(* IEC 61131-3 sources: TA/Tests/RetainTest/Man (part 20) *)

    RETAINTEST_NONRETAIN_STRUCTUREARRAYARRAY.ARRAYARRAY_USINT[2][0] := RETAINTEST_NONRETAIN_STRUCTUREARRAYARRAY.ARRAYARRAY_USINT[2][0] + 1;
    RETAINTEST_NONRETAIN_STRUCTUREARRAYARRAY.ARRAYARRAY_USINT[2][1] := RETAINTEST_NONRETAIN_STRUCTUREARRAYARRAY.ARRAYARRAY_USINT[2][1] + 1;
    RETAINTEST_NONRETAIN_STRUCTUREARRAYARRAY.ARRAYARRAY_USINT[2][2] := RETAINTEST_NONRETAIN_STRUCTUREARRAYARRAY.ARRAYARRAY_USINT[2][2] + 1;
    RETAINTEST_NONRETAIN_STRUCTUREARRAYARRAY.ARRAYARRAY_USINT[2][3] := RETAINTEST_NONRETAIN_STRUCTUREARRAYARRAY.ARRAYARRAY_USINT[2][3] + 1;
    RETAINTEST_NONRETAIN_STRUCTUREARRAYARRAY.ARRAYARRAY_USINT[2][4] := RETAINTEST_NONRETAIN_STRUCTUREARRAYARRAY.ARRAYARRAY_USINT[2][4] + 1;
    RETAINTEST_NONRETAIN_STRUCTUREARRAYARRAY.ARRAYARRAY_USINT[2][5] := RETAINTEST_NONRETAIN_STRUCTUREARRAYARRAY.ARRAYARRAY_USINT[2][5] + 1;
    RETAINTEST_NONRETAIN_STRUCTUREARRAYARRAY.ARRAYARRAY_USINT[2][6] := RETAINTEST_NONRETAIN_STRUCTUREARRAYARRAY.ARRAYARRAY_USINT[2][6] + 1;
    RETAINTEST_NONRETAIN_STRUCTUREARRAYARRAY.ARRAYARRAY_USINT[2][7] := RETAINTEST_NONRETAIN_STRUCTUREARRAYARRAY.ARRAYARRAY_USINT[2][7] + 1;
    RETAINTEST_NONRETAIN_STRUCTUREARRAYARRAY.ARRAYARRAY_USINT[2][8] := RETAINTEST_NONRETAIN_STRUCTUREARRAYARRAY.ARRAYARRAY_USINT[2][8] + 1;
    RETAINTEST_NONRETAIN_STRUCTUREARRAYARRAY.ARRAYARRAY_USINT[2][9] := RETAINTEST_NONRETAIN_STRUCTUREARRAYARRAY.ARRAYARRAY_USINT[2][9] + 1;

    RETAINTEST_NONRETAIN_STRUCTUREARRAYARRAY.ARRAYARRAY_USINT[3][0] := RETAINTEST_NONRETAIN_STRUCTUREARRAYARRAY.ARRAYARRAY_USINT[3][0] + 1;
    RETAINTEST_NONRETAIN_STRUCTUREARRAYARRAY.ARRAYARRAY_USINT[3][1] := RETAINTEST_NONRETAIN_STRUCTUREARRAYARRAY.ARRAYARRAY_USINT[3][1] + 1;
    RETAINTEST_NONRETAIN_STRUCTUREARRAYARRAY.ARRAYARRAY_USINT[3][2] := RETAINTEST_NONRETAIN_STRUCTUREARRAYARRAY.ARRAYARRAY_USINT[3][2] + 1;
    RETAINTEST_NONRETAIN_STRUCTUREARRAYARRAY.ARRAYARRAY_USINT[3][3] := RETAINTEST_NONRETAIN_STRUCTUREARRAYARRAY.ARRAYARRAY_USINT[3][3] + 1;
    RETAINTEST_NONRETAIN_STRUCTUREARRAYARRAY.ARRAYARRAY_USINT[3][4] := RETAINTEST_NONRETAIN_STRUCTUREARRAYARRAY.ARRAYARRAY_USINT[3][4] + 1;
    RETAINTEST_NONRETAIN_STRUCTUREARRAYARRAY.ARRAYARRAY_USINT[3][5] := RETAINTEST_NONRETAIN_STRUCTUREARRAYARRAY.ARRAYARRAY_USINT[3][5] + 1;
    RETAINTEST_NONRETAIN_STRUCTUREARRAYARRAY.ARRAYARRAY_USINT[3][6] := RETAINTEST_NONRETAIN_STRUCTUREARRAYARRAY.ARRAYARRAY_USINT[3][6] + 1;
    RETAINTEST_NONRETAIN_STRUCTUREARRAYARRAY.ARRAYARRAY_USINT[3][7] := RETAINTEST_NONRETAIN_STRUCTUREARRAYARRAY.ARRAYARRAY_USINT[3][7] + 1;
    RETAINTEST_NONRETAIN_STRUCTUREARRAYARRAY.ARRAYARRAY_USINT[3][8] := RETAINTEST_NONRETAIN_STRUCTUREARRAYARRAY.ARRAYARRAY_USINT[3][8] + 1;
    RETAINTEST_NONRETAIN_STRUCTUREARRAYARRAY.ARRAYARRAY_USINT[3][9] := RETAINTEST_NONRETAIN_STRUCTUREARRAYARRAY.ARRAYARRAY_USINT[3][9] + 1;

    RETAINTEST_NONRETAIN_STRUCTUREARRAYARRAY.ARRAYARRAY_USINT[4][0] := RETAINTEST_NONRETAIN_STRUCTUREARRAYARRAY.ARRAYARRAY_USINT[4][0] + 1;
    RETAINTEST_NONRETAIN_STRUCTUREARRAYARRAY.ARRAYARRAY_USINT[4][1] := RETAINTEST_NONRETAIN_STRUCTUREARRAYARRAY.ARRAYARRAY_USINT[4][1] + 1;
    RETAINTEST_NONRETAIN_STRUCTUREARRAYARRAY.ARRAYARRAY_USINT[4][2] := RETAINTEST_NONRETAIN_STRUCTUREARRAYARRAY.ARRAYARRAY_USINT[4][2] + 1;
    RETAINTEST_NONRETAIN_STRUCTUREARRAYARRAY.ARRAYARRAY_USINT[4][3] := RETAINTEST_NONRETAIN_STRUCTUREARRAYARRAY.ARRAYARRAY_USINT[4][3] + 1;
    RETAINTEST_NONRETAIN_STRUCTUREARRAYARRAY.ARRAYARRAY_USINT[4][4] := RETAINTEST_NONRETAIN_STRUCTUREARRAYARRAY.ARRAYARRAY_USINT[4][4] + 1;
    RETAINTEST_NONRETAIN_STRUCTUREARRAYARRAY.ARRAYARRAY_USINT[4][5] := RETAINTEST_NONRETAIN_STRUCTUREARRAYARRAY.ARRAYARRAY_USINT[4][5] + 1;
    RETAINTEST_NONRETAIN_STRUCTUREARRAYARRAY.ARRAYARRAY_USINT[4][6] := RETAINTEST_NONRETAIN_STRUCTUREARRAYARRAY.ARRAYARRAY_USINT[4][6] + 1;
    RETAINTEST_NONRETAIN_STRUCTUREARRAYARRAY.ARRAYARRAY_USINT[4][7] := RETAINTEST_NONRETAIN_STRUCTUREARRAYARRAY.ARRAYARRAY_USINT[4][7] + 1;
    RETAINTEST_NONRETAIN_STRUCTUREARRAYARRAY.ARRAYARRAY_USINT[4][8] := RETAINTEST_NONRETAIN_STRUCTUREARRAYARRAY.ARRAYARRAY_USINT[4][8] + 1;
    RETAINTEST_NONRETAIN_STRUCTUREARRAYARRAY.ARRAYARRAY_USINT[4][9] := RETAINTEST_NONRETAIN_STRUCTUREARRAYARRAY.ARRAYARRAY_USINT[4][9] + 1;

    RETAINTEST_NONRETAIN_STRUCTUREARRAYARRAY.ARRAYARRAY_USINT[5][0] := RETAINTEST_NONRETAIN_STRUCTUREARRAYARRAY.ARRAYARRAY_USINT[5][0] + 1;
    RETAINTEST_NONRETAIN_STRUCTUREARRAYARRAY.ARRAYARRAY_USINT[5][1] := RETAINTEST_NONRETAIN_STRUCTUREARRAYARRAY.ARRAYARRAY_USINT[5][1] + 1;
    RETAINTEST_NONRETAIN_STRUCTUREARRAYARRAY.ARRAYARRAY_USINT[5][2] := RETAINTEST_NONRETAIN_STRUCTUREARRAYARRAY.ARRAYARRAY_USINT[5][2] + 1;
    RETAINTEST_NONRETAIN_STRUCTUREARRAYARRAY.ARRAYARRAY_USINT[5][3] := RETAINTEST_NONRETAIN_STRUCTUREARRAYARRAY.ARRAYARRAY_USINT[5][3] + 1;
    RETAINTEST_NONRETAIN_STRUCTUREARRAYARRAY.ARRAYARRAY_USINT[5][4] := RETAINTEST_NONRETAIN_STRUCTUREARRAYARRAY.ARRAYARRAY_USINT[5][4] + 1;
    RETAINTEST_NONRETAIN_STRUCTUREARRAYARRAY.ARRAYARRAY_USINT[5][5] := RETAINTEST_NONRETAIN_STRUCTUREARRAYARRAY.ARRAYARRAY_USINT[5][5] + 1;
    RETAINTEST_NONRETAIN_STRUCTUREARRAYARRAY.ARRAYARRAY_USINT[5][6] := RETAINTEST_NONRETAIN_STRUCTUREARRAYARRAY.ARRAYARRAY_USINT[5][6] + 1;
    RETAINTEST_NONRETAIN_STRUCTUREARRAYARRAY.ARRAYARRAY_USINT[5][7] := RETAINTEST_NONRETAIN_STRUCTUREARRAYARRAY.ARRAYARRAY_USINT[5][7] + 1;
    RETAINTEST_NONRETAIN_STRUCTUREARRAYARRAY.ARRAYARRAY_USINT[5][8] := RETAINTEST_NONRETAIN_STRUCTUREARRAYARRAY.ARRAYARRAY_USINT[5][8] + 1;
    RETAINTEST_NONRETAIN_STRUCTUREARRAYARRAY.ARRAYARRAY_USINT[5][9] := RETAINTEST_NONRETAIN_STRUCTUREARRAYARRAY.ARRAYARRAY_USINT[5][9] + 1;

    RETAINTEST_NONRETAIN_STRUCTUREARRAYARRAY.ARRAYARRAY_USINT[6][0] := RETAINTEST_NONRETAIN_STRUCTUREARRAYARRAY.ARRAYARRAY_USINT[6][0] + 1;
    RETAINTEST_NONRETAIN_STRUCTUREARRAYARRAY.ARRAYARRAY_USINT[6][1] := RETAINTEST_NONRETAIN_STRUCTUREARRAYARRAY.ARRAYARRAY_USINT[6][1] + 1;
    RETAINTEST_NONRETAIN_STRUCTUREARRAYARRAY.ARRAYARRAY_USINT[6][2] := RETAINTEST_NONRETAIN_STRUCTUREARRAYARRAY.ARRAYARRAY_USINT[6][2] + 1;
    RETAINTEST_NONRETAIN_STRUCTUREARRAYARRAY.ARRAYARRAY_USINT[6][3] := RETAINTEST_NONRETAIN_STRUCTUREARRAYARRAY.ARRAYARRAY_USINT[6][3] + 1;
    RETAINTEST_NONRETAIN_STRUCTUREARRAYARRAY.ARRAYARRAY_USINT[6][4] := RETAINTEST_NONRETAIN_STRUCTUREARRAYARRAY.ARRAYARRAY_USINT[6][4] + 1;
    RETAINTEST_NONRETAIN_STRUCTUREARRAYARRAY.ARRAYARRAY_USINT[6][5] := RETAINTEST_NONRETAIN_STRUCTUREARRAYARRAY.ARRAYARRAY_USINT[6][5] + 1;
    RETAINTEST_NONRETAIN_STRUCTUREARRAYARRAY.ARRAYARRAY_USINT[6][6] := RETAINTEST_NONRETAIN_STRUCTUREARRAYARRAY.ARRAYARRAY_USINT[6][6] + 1;
    RETAINTEST_NONRETAIN_STRUCTUREARRAYARRAY.ARRAYARRAY_USINT[6][7] := RETAINTEST_NONRETAIN_STRUCTUREARRAYARRAY.ARRAYARRAY_USINT[6][7] + 1;
    RETAINTEST_NONRETAIN_STRUCTUREARRAYARRAY.ARRAYARRAY_USINT[6][8] := RETAINTEST_NONRETAIN_STRUCTUREARRAYARRAY.ARRAYARRAY_USINT[6][8] + 1;
    RETAINTEST_NONRETAIN_STRUCTUREARRAYARRAY.ARRAYARRAY_USINT[6][9] := RETAINTEST_NONRETAIN_STRUCTUREARRAYARRAY.ARRAYARRAY_USINT[6][9] + 1;

    RETAINTEST_NONRETAIN_STRUCTUREARRAYARRAY.ARRAYARRAY_USINT[7][0] := RETAINTEST_NONRETAIN_STRUCTUREARRAYARRAY.ARRAYARRAY_USINT[6][0];
    RETAINTEST_NONRETAIN_STRUCTUREARRAYARRAY.ARRAYARRAY_USINT[7][1] := RETAINTEST_NONRETAIN_STRUCTUREARRAYARRAY.ARRAYARRAY_USINT[6][1];
    RETAINTEST_NONRETAIN_STRUCTUREARRAYARRAY.ARRAYARRAY_USINT[7][2] := RETAINTEST_NONRETAIN_STRUCTUREARRAYARRAY.ARRAYARRAY_USINT[6][2];
    RETAINTEST_NONRETAIN_STRUCTUREARRAYARRAY.ARRAYARRAY_USINT[7][3] := RETAINTEST_NONRETAIN_STRUCTUREARRAYARRAY.ARRAYARRAY_USINT[6][3];
    RETAINTEST_NONRETAIN_STRUCTUREARRAYARRAY.ARRAYARRAY_USINT[7][4] := RETAINTEST_NONRETAIN_STRUCTUREARRAYARRAY.ARRAYARRAY_USINT[6][4];
    RETAINTEST_NONRETAIN_STRUCTUREARRAYARRAY.ARRAYARRAY_USINT[7][5] := RETAINTEST_NONRETAIN_STRUCTUREARRAYARRAY.ARRAYARRAY_USINT[6][5];
    RETAINTEST_NONRETAIN_STRUCTUREARRAYARRAY.ARRAYARRAY_USINT[7][6] := RETAINTEST_NONRETAIN_STRUCTUREARRAYARRAY.ARRAYARRAY_USINT[6][6];
    RETAINTEST_NONRETAIN_STRUCTUREARRAYARRAY.ARRAYARRAY_USINT[7][7] := RETAINTEST_NONRETAIN_STRUCTUREARRAYARRAY.ARRAYARRAY_USINT[6][7];
    RETAINTEST_NONRETAIN_STRUCTUREARRAYARRAY.ARRAYARRAY_USINT[7][8] := RETAINTEST_NONRETAIN_STRUCTUREARRAYARRAY.ARRAYARRAY_USINT[6][8];
    RETAINTEST_NONRETAIN_STRUCTUREARRAYARRAY.ARRAYARRAY_USINT[7][9] := RETAINTEST_NONRETAIN_STRUCTUREARRAYARRAY.ARRAYARRAY_USINT[6][9];

    RETAINTEST_NONRETAIN_STRUCTUREARRAYARRAY.ARRAYARRAY_WORD[0][0] := RETAINTEST_NONRETAIN_STRUCTUREARRAYARRAY.ARRAYARRAY_WORD[0][0] + 1;
    RETAINTEST_NONRETAIN_STRUCTUREARRAYARRAY.ARRAYARRAY_WORD[0][1] := RETAINTEST_NONRETAIN_STRUCTUREARRAYARRAY.ARRAYARRAY_WORD[0][1] + 1;
    RETAINTEST_NONRETAIN_STRUCTUREARRAYARRAY.ARRAYARRAY_WORD[0][2] := RETAINTEST_NONRETAIN_STRUCTUREARRAYARRAY.ARRAYARRAY_WORD[0][2] + 1;
    RETAINTEST_NONRETAIN_STRUCTUREARRAYARRAY.ARRAYARRAY_WORD[0][3] := RETAINTEST_NONRETAIN_STRUCTUREARRAYARRAY.ARRAYARRAY_WORD[0][3] + 1;
    RETAINTEST_NONRETAIN_STRUCTUREARRAYARRAY.ARRAYARRAY_WORD[0][4] := RETAINTEST_NONRETAIN_STRUCTUREARRAYARRAY.ARRAYARRAY_WORD[0][4] + 1;
    RETAINTEST_NONRETAIN_STRUCTUREARRAYARRAY.ARRAYARRAY_WORD[0][5] := RETAINTEST_NONRETAIN_STRUCTUREARRAYARRAY.ARRAYARRAY_WORD[0][5] + 1;
    RETAINTEST_NONRETAIN_STRUCTUREARRAYARRAY.ARRAYARRAY_WORD[0][6] := RETAINTEST_NONRETAIN_STRUCTUREARRAYARRAY.ARRAYARRAY_WORD[0][6] + 1;
    RETAINTEST_NONRETAIN_STRUCTUREARRAYARRAY.ARRAYARRAY_WORD[0][7] := RETAINTEST_NONRETAIN_STRUCTUREARRAYARRAY.ARRAYARRAY_WORD[0][7] + 1;
    RETAINTEST_NONRETAIN_STRUCTUREARRAYARRAY.ARRAYARRAY_WORD[0][8] := RETAINTEST_NONRETAIN_STRUCTUREARRAYARRAY.ARRAYARRAY_WORD[0][6];
    RETAINTEST_NONRETAIN_STRUCTUREARRAYARRAY.ARRAYARRAY_WORD[0][9] := RETAINTEST_NONRETAIN_STRUCTUREARRAYARRAY.ARRAYARRAY_WORD[0][7];

    RETAINTEST_NONRETAIN_STRUCTUREARRAYARRAY.ARRAYARRAY_WORD[1][0] := RETAINTEST_NONRETAIN_STRUCTUREARRAYARRAY.ARRAYARRAY_WORD[1][0] + 1;
    RETAINTEST_NONRETAIN_STRUCTUREARRAYARRAY.ARRAYARRAY_WORD[1][1] := RETAINTEST_NONRETAIN_STRUCTUREARRAYARRAY.ARRAYARRAY_WORD[1][1] + 1;
    RETAINTEST_NONRETAIN_STRUCTUREARRAYARRAY.ARRAYARRAY_WORD[1][2] := RETAINTEST_NONRETAIN_STRUCTUREARRAYARRAY.ARRAYARRAY_WORD[1][2] + 1;
    RETAINTEST_NONRETAIN_STRUCTUREARRAYARRAY.ARRAYARRAY_WORD[1][3] := RETAINTEST_NONRETAIN_STRUCTUREARRAYARRAY.ARRAYARRAY_WORD[1][3] + 1;
    RETAINTEST_NONRETAIN_STRUCTUREARRAYARRAY.ARRAYARRAY_WORD[1][4] := RETAINTEST_NONRETAIN_STRUCTUREARRAYARRAY.ARRAYARRAY_WORD[1][4] + 1;
    RETAINTEST_NONRETAIN_STRUCTUREARRAYARRAY.ARRAYARRAY_WORD[1][5] := RETAINTEST_NONRETAIN_STRUCTUREARRAYARRAY.ARRAYARRAY_WORD[1][5] + 1;
    RETAINTEST_NONRETAIN_STRUCTUREARRAYARRAY.ARRAYARRAY_WORD[1][6] := RETAINTEST_NONRETAIN_STRUCTUREARRAYARRAY.ARRAYARRAY_WORD[1][6] + 1;
    RETAINTEST_NONRETAIN_STRUCTUREARRAYARRAY.ARRAYARRAY_WORD[1][7] := RETAINTEST_NONRETAIN_STRUCTUREARRAYARRAY.ARRAYARRAY_WORD[1][7] + 1;
    RETAINTEST_NONRETAIN_STRUCTUREARRAYARRAY.ARRAYARRAY_WORD[1][8] := RETAINTEST_NONRETAIN_STRUCTUREARRAYARRAY.ARRAYARRAY_WORD[1][6];
    RETAINTEST_NONRETAIN_STRUCTUREARRAYARRAY.ARRAYARRAY_WORD[1][9] := RETAINTEST_NONRETAIN_STRUCTUREARRAYARRAY.ARRAYARRAY_WORD[1][7];

    RETAINTEST_NONRETAIN_STRUCTUREARRAYARRAY.ARRAYARRAY_WORD[2][0] := RETAINTEST_NONRETAIN_STRUCTUREARRAYARRAY.ARRAYARRAY_WORD[2][0] + 1;
    RETAINTEST_NONRETAIN_STRUCTUREARRAYARRAY.ARRAYARRAY_WORD[2][1] := RETAINTEST_NONRETAIN_STRUCTUREARRAYARRAY.ARRAYARRAY_WORD[2][1] + 1;
    RETAINTEST_NONRETAIN_STRUCTUREARRAYARRAY.ARRAYARRAY_WORD[2][2] := RETAINTEST_NONRETAIN_STRUCTUREARRAYARRAY.ARRAYARRAY_WORD[2][2] + 1;
    RETAINTEST_NONRETAIN_STRUCTUREARRAYARRAY.ARRAYARRAY_WORD[2][3] := RETAINTEST_NONRETAIN_STRUCTUREARRAYARRAY.ARRAYARRAY_WORD[2][3] + 1;
    RETAINTEST_NONRETAIN_STRUCTUREARRAYARRAY.ARRAYARRAY_WORD[2][4] := RETAINTEST_NONRETAIN_STRUCTUREARRAYARRAY.ARRAYARRAY_WORD[2][4] + 1;
    RETAINTEST_NONRETAIN_STRUCTUREARRAYARRAY.ARRAYARRAY_WORD[2][5] := RETAINTEST_NONRETAIN_STRUCTUREARRAYARRAY.ARRAYARRAY_WORD[2][5] + 1;
    RETAINTEST_NONRETAIN_STRUCTUREARRAYARRAY.ARRAYARRAY_WORD[2][6] := RETAINTEST_NONRETAIN_STRUCTUREARRAYARRAY.ARRAYARRAY_WORD[2][6] + 1;
    RETAINTEST_NONRETAIN_STRUCTUREARRAYARRAY.ARRAYARRAY_WORD[2][7] := RETAINTEST_NONRETAIN_STRUCTUREARRAYARRAY.ARRAYARRAY_WORD[2][7] + 1;
    RETAINTEST_NONRETAIN_STRUCTUREARRAYARRAY.ARRAYARRAY_WORD[2][8] := RETAINTEST_NONRETAIN_STRUCTUREARRAYARRAY.ARRAYARRAY_WORD[2][8] + 1;
    RETAINTEST_NONRETAIN_STRUCTUREARRAYARRAY.ARRAYARRAY_WORD[2][9] := RETAINTEST_NONRETAIN_STRUCTUREARRAYARRAY.ARRAYARRAY_WORD[2][9] + 1;

    RETAINTEST_NONRETAIN_STRUCTUREARRAYARRAY.ARRAYARRAY_WORD[3][0] := RETAINTEST_NONRETAIN_STRUCTUREARRAYARRAY.ARRAYARRAY_WORD[3][0] + 1;
    RETAINTEST_NONRETAIN_STRUCTUREARRAYARRAY.ARRAYARRAY_WORD[3][1] := RETAINTEST_NONRETAIN_STRUCTUREARRAYARRAY.ARRAYARRAY_WORD[3][1] + 1;
    RETAINTEST_NONRETAIN_STRUCTUREARRAYARRAY.ARRAYARRAY_WORD[3][2] := RETAINTEST_NONRETAIN_STRUCTUREARRAYARRAY.ARRAYARRAY_WORD[3][2] + 1;
    RETAINTEST_NONRETAIN_STRUCTUREARRAYARRAY.ARRAYARRAY_WORD[3][3] := RETAINTEST_NONRETAIN_STRUCTUREARRAYARRAY.ARRAYARRAY_WORD[3][3] + 1;
    RETAINTEST_NONRETAIN_STRUCTUREARRAYARRAY.ARRAYARRAY_WORD[3][4] := RETAINTEST_NONRETAIN_STRUCTUREARRAYARRAY.ARRAYARRAY_WORD[3][4] + 1;
    RETAINTEST_NONRETAIN_STRUCTUREARRAYARRAY.ARRAYARRAY_WORD[3][5] := RETAINTEST_NONRETAIN_STRUCTUREARRAYARRAY.ARRAYARRAY_WORD[3][5] + 1;
    RETAINTEST_NONRETAIN_STRUCTUREARRAYARRAY.ARRAYARRAY_WORD[3][6] := RETAINTEST_NONRETAIN_STRUCTUREARRAYARRAY.ARRAYARRAY_WORD[3][6] + 1;
    RETAINTEST_NONRETAIN_STRUCTUREARRAYARRAY.ARRAYARRAY_WORD[3][7] := RETAINTEST_NONRETAIN_STRUCTUREARRAYARRAY.ARRAYARRAY_WORD[3][7] + 1;
    RETAINTEST_NONRETAIN_STRUCTUREARRAYARRAY.ARRAYARRAY_WORD[3][8] := RETAINTEST_NONRETAIN_STRUCTUREARRAYARRAY.ARRAYARRAY_WORD[3][8] + 1;
    RETAINTEST_NONRETAIN_STRUCTUREARRAYARRAY.ARRAYARRAY_WORD[3][9] := RETAINTEST_NONRETAIN_STRUCTUREARRAYARRAY.ARRAYARRAY_WORD[3][9] + 1;

    RETAINTEST_NONRETAIN_STRUCTUREARRAYARRAY.ARRAYARRAY_WORD[4][0] := RETAINTEST_NONRETAIN_STRUCTUREARRAYARRAY.ARRAYARRAY_WORD[4][0] + 1;
    RETAINTEST_NONRETAIN_STRUCTUREARRAYARRAY.ARRAYARRAY_WORD[4][1] := RETAINTEST_NONRETAIN_STRUCTUREARRAYARRAY.ARRAYARRAY_WORD[4][1] + 1;
    RETAINTEST_NONRETAIN_STRUCTUREARRAYARRAY.ARRAYARRAY_WORD[4][2] := RETAINTEST_NONRETAIN_STRUCTUREARRAYARRAY.ARRAYARRAY_WORD[4][2] + 1;
    RETAINTEST_NONRETAIN_STRUCTUREARRAYARRAY.ARRAYARRAY_WORD[4][3] := RETAINTEST_NONRETAIN_STRUCTUREARRAYARRAY.ARRAYARRAY_WORD[4][3] + 1;
    RETAINTEST_NONRETAIN_STRUCTUREARRAYARRAY.ARRAYARRAY_WORD[4][4] := RETAINTEST_NONRETAIN_STRUCTUREARRAYARRAY.ARRAYARRAY_WORD[4][4] + 1;
    RETAINTEST_NONRETAIN_STRUCTUREARRAYARRAY.ARRAYARRAY_WORD[4][5] := RETAINTEST_NONRETAIN_STRUCTUREARRAYARRAY.ARRAYARRAY_WORD[4][5] + 1;
    RETAINTEST_NONRETAIN_STRUCTUREARRAYARRAY.ARRAYARRAY_WORD[4][6] := RETAINTEST_NONRETAIN_STRUCTUREARRAYARRAY.ARRAYARRAY_WORD[4][6] + 1;
    RETAINTEST_NONRETAIN_STRUCTUREARRAYARRAY.ARRAYARRAY_WORD[4][7] := RETAINTEST_NONRETAIN_STRUCTUREARRAYARRAY.ARRAYARRAY_WORD[4][7] + 1;
    RETAINTEST_NONRETAIN_STRUCTUREARRAYARRAY.ARRAYARRAY_WORD[4][8] := RETAINTEST_NONRETAIN_STRUCTUREARRAYARRAY.ARRAYARRAY_WORD[4][8] + 1;
    RETAINTEST_NONRETAIN_STRUCTUREARRAYARRAY.ARRAYARRAY_WORD[4][9] := RETAINTEST_NONRETAIN_STRUCTUREARRAYARRAY.ARRAYARRAY_WORD[4][9] + 1;

    RETAINTEST_NONRETAIN_STRUCTUREARRAYARRAY.ARRAYARRAY_WORD[5][0] := RETAINTEST_NONRETAIN_STRUCTUREARRAYARRAY.ARRAYARRAY_WORD[5][0] + 1;
    RETAINTEST_NONRETAIN_STRUCTUREARRAYARRAY.ARRAYARRAY_WORD[5][1] := RETAINTEST_NONRETAIN_STRUCTUREARRAYARRAY.ARRAYARRAY_WORD[5][1] + 1;
    RETAINTEST_NONRETAIN_STRUCTUREARRAYARRAY.ARRAYARRAY_WORD[5][2] := RETAINTEST_NONRETAIN_STRUCTUREARRAYARRAY.ARRAYARRAY_WORD[5][2] + 1;
    RETAINTEST_NONRETAIN_STRUCTUREARRAYARRAY.ARRAYARRAY_WORD[5][3] := RETAINTEST_NONRETAIN_STRUCTUREARRAYARRAY.ARRAYARRAY_WORD[5][3] + 1;
    RETAINTEST_NONRETAIN_STRUCTUREARRAYARRAY.ARRAYARRAY_WORD[5][4] := RETAINTEST_NONRETAIN_STRUCTUREARRAYARRAY.ARRAYARRAY_WORD[5][4] + 1;
    RETAINTEST_NONRETAIN_STRUCTUREARRAYARRAY.ARRAYARRAY_WORD[5][5] := RETAINTEST_NONRETAIN_STRUCTUREARRAYARRAY.ARRAYARRAY_WORD[5][5] + 1;
    RETAINTEST_NONRETAIN_STRUCTUREARRAYARRAY.ARRAYARRAY_WORD[5][6] := RETAINTEST_NONRETAIN_STRUCTUREARRAYARRAY.ARRAYARRAY_WORD[5][6] + 1;
    RETAINTEST_NONRETAIN_STRUCTUREARRAYARRAY.ARRAYARRAY_WORD[5][7] := RETAINTEST_NONRETAIN_STRUCTUREARRAYARRAY.ARRAYARRAY_WORD[5][7] + 1;
    RETAINTEST_NONRETAIN_STRUCTUREARRAYARRAY.ARRAYARRAY_WORD[5][8] := RETAINTEST_NONRETAIN_STRUCTUREARRAYARRAY.ARRAYARRAY_WORD[5][8] + 1;
    RETAINTEST_NONRETAIN_STRUCTUREARRAYARRAY.ARRAYARRAY_WORD[5][9] := RETAINTEST_NONRETAIN_STRUCTUREARRAYARRAY.ARRAYARRAY_WORD[5][9] + 1;

    RETAINTEST_NONRETAIN_STRUCTUREARRAYARRAY.ARRAYARRAY_WORD[6][0] := RETAINTEST_NONRETAIN_STRUCTUREARRAYARRAY.ARRAYARRAY_WORD[6][0] + 1;
    RETAINTEST_NONRETAIN_STRUCTUREARRAYARRAY.ARRAYARRAY_WORD[6][1] := RETAINTEST_NONRETAIN_STRUCTUREARRAYARRAY.ARRAYARRAY_WORD[6][1] + 1;
    RETAINTEST_NONRETAIN_STRUCTUREARRAYARRAY.ARRAYARRAY_WORD[6][2] := RETAINTEST_NONRETAIN_STRUCTUREARRAYARRAY.ARRAYARRAY_WORD[6][2] + 1;
    RETAINTEST_NONRETAIN_STRUCTUREARRAYARRAY.ARRAYARRAY_WORD[6][3] := RETAINTEST_NONRETAIN_STRUCTUREARRAYARRAY.ARRAYARRAY_WORD[6][3] + 1;
    RETAINTEST_NONRETAIN_STRUCTUREARRAYARRAY.ARRAYARRAY_WORD[6][4] := RETAINTEST_NONRETAIN_STRUCTUREARRAYARRAY.ARRAYARRAY_WORD[6][4] + 1;
    RETAINTEST_NONRETAIN_STRUCTUREARRAYARRAY.ARRAYARRAY_WORD[6][5] := RETAINTEST_NONRETAIN_STRUCTUREARRAYARRAY.ARRAYARRAY_WORD[6][5] + 1;
    RETAINTEST_NONRETAIN_STRUCTUREARRAYARRAY.ARRAYARRAY_WORD[6][6] := RETAINTEST_NONRETAIN_STRUCTUREARRAYARRAY.ARRAYARRAY_WORD[6][6] + 1;
    RETAINTEST_NONRETAIN_STRUCTUREARRAYARRAY.ARRAYARRAY_WORD[6][7] := RETAINTEST_NONRETAIN_STRUCTUREARRAYARRAY.ARRAYARRAY_WORD[6][7] + 1;
    RETAINTEST_NONRETAIN_STRUCTUREARRAYARRAY.ARRAYARRAY_WORD[6][8] := RETAINTEST_NONRETAIN_STRUCTUREARRAYARRAY.ARRAYARRAY_WORD[6][8] + 1;
    RETAINTEST_NONRETAIN_STRUCTUREARRAYARRAY.ARRAYARRAY_WORD[6][9] := RETAINTEST_NONRETAIN_STRUCTUREARRAYARRAY.ARRAYARRAY_WORD[6][9] + 1;

    RETAINTEST_NONRETAIN_STRUCTUREARRAYARRAY.ARRAYARRAY_WORD[7][0] := RETAINTEST_NONRETAIN_STRUCTUREARRAYARRAY.ARRAYARRAY_WORD[6][0];
    RETAINTEST_NONRETAIN_STRUCTUREARRAYARRAY.ARRAYARRAY_WORD[7][1] := RETAINTEST_NONRETAIN_STRUCTUREARRAYARRAY.ARRAYARRAY_WORD[6][1];
    RETAINTEST_NONRETAIN_STRUCTUREARRAYARRAY.ARRAYARRAY_WORD[7][2] := RETAINTEST_NONRETAIN_STRUCTUREARRAYARRAY.ARRAYARRAY_WORD[6][2];
    RETAINTEST_NONRETAIN_STRUCTUREARRAYARRAY.ARRAYARRAY_WORD[7][3] := RETAINTEST_NONRETAIN_STRUCTUREARRAYARRAY.ARRAYARRAY_WORD[6][3];
    RETAINTEST_NONRETAIN_STRUCTUREARRAYARRAY.ARRAYARRAY_WORD[7][4] := RETAINTEST_NONRETAIN_STRUCTUREARRAYARRAY.ARRAYARRAY_WORD[6][4];
    RETAINTEST_NONRETAIN_STRUCTUREARRAYARRAY.ARRAYARRAY_WORD[7][5] := RETAINTEST_NONRETAIN_STRUCTUREARRAYARRAY.ARRAYARRAY_WORD[6][5];
    RETAINTEST_NONRETAIN_STRUCTUREARRAYARRAY.ARRAYARRAY_WORD[7][6] := RETAINTEST_NONRETAIN_STRUCTUREARRAYARRAY.ARRAYARRAY_WORD[6][6];
    RETAINTEST_NONRETAIN_STRUCTUREARRAYARRAY.ARRAYARRAY_WORD[7][7] := RETAINTEST_NONRETAIN_STRUCTUREARRAYARRAY.ARRAYARRAY_WORD[6][7];
    RETAINTEST_NONRETAIN_STRUCTUREARRAYARRAY.ARRAYARRAY_WORD[7][8] := RETAINTEST_NONRETAIN_STRUCTUREARRAYARRAY.ARRAYARRAY_WORD[6][8];
    RETAINTEST_NONRETAIN_STRUCTUREARRAYARRAY.ARRAYARRAY_WORD[7][9] := RETAINTEST_NONRETAIN_STRUCTUREARRAYARRAY.ARRAYARRAY_WORD[6][9];

    RETAINTEST_AUTO_STRUCTUREARRAYARRAY.ARRAYARRAY_BOOL[0][0] := NOT RETAINTEST_AUTO_STRUCTUREARRAYARRAY.ARRAYARRAY_BOOL[0][0];
    RETAINTEST_AUTO_STRUCTUREARRAYARRAY.ARRAYARRAY_BOOL[0][1] := NOT RETAINTEST_AUTO_STRUCTUREARRAYARRAY.ARRAYARRAY_BOOL[0][1];
    RETAINTEST_AUTO_STRUCTUREARRAYARRAY.ARRAYARRAY_BOOL[0][2] := NOT RETAINTEST_AUTO_STRUCTUREARRAYARRAY.ARRAYARRAY_BOOL[0][2];
    RETAINTEST_AUTO_STRUCTUREARRAYARRAY.ARRAYARRAY_BOOL[0][3] := NOT RETAINTEST_AUTO_STRUCTUREARRAYARRAY.ARRAYARRAY_BOOL[0][3];
    RETAINTEST_AUTO_STRUCTUREARRAYARRAY.ARRAYARRAY_BOOL[0][4] := NOT RETAINTEST_AUTO_STRUCTUREARRAYARRAY.ARRAYARRAY_BOOL[0][4];
    RETAINTEST_AUTO_STRUCTUREARRAYARRAY.ARRAYARRAY_BOOL[0][5] := NOT RETAINTEST_AUTO_STRUCTUREARRAYARRAY.ARRAYARRAY_BOOL[0][5];
    RETAINTEST_AUTO_STRUCTUREARRAYARRAY.ARRAYARRAY_BOOL[0][6] := NOT RETAINTEST_AUTO_STRUCTUREARRAYARRAY.ARRAYARRAY_BOOL[0][6];
    RETAINTEST_AUTO_STRUCTUREARRAYARRAY.ARRAYARRAY_BOOL[0][7] := NOT RETAINTEST_AUTO_STRUCTUREARRAYARRAY.ARRAYARRAY_BOOL[0][7];
    RETAINTEST_AUTO_STRUCTUREARRAYARRAY.ARRAYARRAY_BOOL[0][8] := RETAINTEST_AUTO_STRUCTUREARRAYARRAY.ARRAYARRAY_BOOL[0][6];
    RETAINTEST_AUTO_STRUCTUREARRAYARRAY.ARRAYARRAY_BOOL[0][9] := RETAINTEST_AUTO_STRUCTUREARRAYARRAY.ARRAYARRAY_BOOL[0][7];

    RETAINTEST_AUTO_STRUCTUREARRAYARRAY.ARRAYARRAY_BOOL[1][0] := NOT RETAINTEST_AUTO_STRUCTUREARRAYARRAY.ARRAYARRAY_BOOL[1][0];
    RETAINTEST_AUTO_STRUCTUREARRAYARRAY.ARRAYARRAY_BOOL[1][1] := NOT RETAINTEST_AUTO_STRUCTUREARRAYARRAY.ARRAYARRAY_BOOL[1][1];
    RETAINTEST_AUTO_STRUCTUREARRAYARRAY.ARRAYARRAY_BOOL[1][2] := NOT RETAINTEST_AUTO_STRUCTUREARRAYARRAY.ARRAYARRAY_BOOL[1][2];
    RETAINTEST_AUTO_STRUCTUREARRAYARRAY.ARRAYARRAY_BOOL[1][3] := NOT RETAINTEST_AUTO_STRUCTUREARRAYARRAY.ARRAYARRAY_BOOL[1][3];
    RETAINTEST_AUTO_STRUCTUREARRAYARRAY.ARRAYARRAY_BOOL[1][4] := NOT RETAINTEST_AUTO_STRUCTUREARRAYARRAY.ARRAYARRAY_BOOL[1][4];
    RETAINTEST_AUTO_STRUCTUREARRAYARRAY.ARRAYARRAY_BOOL[1][5] := NOT RETAINTEST_AUTO_STRUCTUREARRAYARRAY.ARRAYARRAY_BOOL[1][5];
    RETAINTEST_AUTO_STRUCTUREARRAYARRAY.ARRAYARRAY_BOOL[1][6] := NOT RETAINTEST_AUTO_STRUCTUREARRAYARRAY.ARRAYARRAY_BOOL[1][6];
    RETAINTEST_AUTO_STRUCTUREARRAYARRAY.ARRAYARRAY_BOOL[1][7] := NOT RETAINTEST_AUTO_STRUCTUREARRAYARRAY.ARRAYARRAY_BOOL[1][7];
    RETAINTEST_AUTO_STRUCTUREARRAYARRAY.ARRAYARRAY_BOOL[1][8] := RETAINTEST_AUTO_STRUCTUREARRAYARRAY.ARRAYARRAY_BOOL[1][6];
    RETAINTEST_AUTO_STRUCTUREARRAYARRAY.ARRAYARRAY_BOOL[1][9] := RETAINTEST_AUTO_STRUCTUREARRAYARRAY.ARRAYARRAY_BOOL[1][7];

    RETAINTEST_AUTO_STRUCTUREARRAYARRAY.ARRAYARRAY_BOOL[2][0] := NOT RETAINTEST_AUTO_STRUCTUREARRAYARRAY.ARRAYARRAY_BOOL[2][0];
    RETAINTEST_AUTO_STRUCTUREARRAYARRAY.ARRAYARRAY_BOOL[2][1] := NOT RETAINTEST_AUTO_STRUCTUREARRAYARRAY.ARRAYARRAY_BOOL[2][1];
    RETAINTEST_AUTO_STRUCTUREARRAYARRAY.ARRAYARRAY_BOOL[2][2] := NOT RETAINTEST_AUTO_STRUCTUREARRAYARRAY.ARRAYARRAY_BOOL[2][2];
    RETAINTEST_AUTO_STRUCTUREARRAYARRAY.ARRAYARRAY_BOOL[2][3] := NOT RETAINTEST_AUTO_STRUCTUREARRAYARRAY.ARRAYARRAY_BOOL[2][3];
    RETAINTEST_AUTO_STRUCTUREARRAYARRAY.ARRAYARRAY_BOOL[2][4] := NOT RETAINTEST_AUTO_STRUCTUREARRAYARRAY.ARRAYARRAY_BOOL[2][4];
    RETAINTEST_AUTO_STRUCTUREARRAYARRAY.ARRAYARRAY_BOOL[2][5] := NOT RETAINTEST_AUTO_STRUCTUREARRAYARRAY.ARRAYARRAY_BOOL[2][5];
    RETAINTEST_AUTO_STRUCTUREARRAYARRAY.ARRAYARRAY_BOOL[2][6] := NOT RETAINTEST_AUTO_STRUCTUREARRAYARRAY.ARRAYARRAY_BOOL[2][6];
    RETAINTEST_AUTO_STRUCTUREARRAYARRAY.ARRAYARRAY_BOOL[2][7] := NOT RETAINTEST_AUTO_STRUCTUREARRAYARRAY.ARRAYARRAY_BOOL[2][7];
    RETAINTEST_AUTO_STRUCTUREARRAYARRAY.ARRAYARRAY_BOOL[2][8] := NOT RETAINTEST_AUTO_STRUCTUREARRAYARRAY.ARRAYARRAY_BOOL[2][8];
    RETAINTEST_AUTO_STRUCTUREARRAYARRAY.ARRAYARRAY_BOOL[2][9] := NOT RETAINTEST_AUTO_STRUCTUREARRAYARRAY.ARRAYARRAY_BOOL[2][9];

    RETAINTEST_AUTO_STRUCTUREARRAYARRAY.ARRAYARRAY_BOOL[3][0] := NOT RETAINTEST_AUTO_STRUCTUREARRAYARRAY.ARRAYARRAY_BOOL[3][0];
    RETAINTEST_AUTO_STRUCTUREARRAYARRAY.ARRAYARRAY_BOOL[3][1] := NOT RETAINTEST_AUTO_STRUCTUREARRAYARRAY.ARRAYARRAY_BOOL[3][1];
    RETAINTEST_AUTO_STRUCTUREARRAYARRAY.ARRAYARRAY_BOOL[3][2] := NOT RETAINTEST_AUTO_STRUCTUREARRAYARRAY.ARRAYARRAY_BOOL[3][2];
    RETAINTEST_AUTO_STRUCTUREARRAYARRAY.ARRAYARRAY_BOOL[3][3] := NOT RETAINTEST_AUTO_STRUCTUREARRAYARRAY.ARRAYARRAY_BOOL[3][3];
    RETAINTEST_AUTO_STRUCTUREARRAYARRAY.ARRAYARRAY_BOOL[3][4] := NOT RETAINTEST_AUTO_STRUCTUREARRAYARRAY.ARRAYARRAY_BOOL[3][4];
    RETAINTEST_AUTO_STRUCTUREARRAYARRAY.ARRAYARRAY_BOOL[3][5] := NOT RETAINTEST_AUTO_STRUCTUREARRAYARRAY.ARRAYARRAY_BOOL[3][5];
    RETAINTEST_AUTO_STRUCTUREARRAYARRAY.ARRAYARRAY_BOOL[3][6] := NOT RETAINTEST_AUTO_STRUCTUREARRAYARRAY.ARRAYARRAY_BOOL[3][6];
    RETAINTEST_AUTO_STRUCTUREARRAYARRAY.ARRAYARRAY_BOOL[3][7] := NOT RETAINTEST_AUTO_STRUCTUREARRAYARRAY.ARRAYARRAY_BOOL[3][7];
    RETAINTEST_AUTO_STRUCTUREARRAYARRAY.ARRAYARRAY_BOOL[3][8] := NOT RETAINTEST_AUTO_STRUCTUREARRAYARRAY.ARRAYARRAY_BOOL[3][8];
    RETAINTEST_AUTO_STRUCTUREARRAYARRAY.ARRAYARRAY_BOOL[3][9] := NOT RETAINTEST_AUTO_STRUCTUREARRAYARRAY.ARRAYARRAY_BOOL[3][9];

    RETAINTEST_AUTO_STRUCTUREARRAYARRAY.ARRAYARRAY_BOOL[4][0] := NOT RETAINTEST_AUTO_STRUCTUREARRAYARRAY.ARRAYARRAY_BOOL[4][0];
    RETAINTEST_AUTO_STRUCTUREARRAYARRAY.ARRAYARRAY_BOOL[4][1] := NOT RETAINTEST_AUTO_STRUCTUREARRAYARRAY.ARRAYARRAY_BOOL[4][1];
    RETAINTEST_AUTO_STRUCTUREARRAYARRAY.ARRAYARRAY_BOOL[4][2] := NOT RETAINTEST_AUTO_STRUCTUREARRAYARRAY.ARRAYARRAY_BOOL[4][2];
    RETAINTEST_AUTO_STRUCTUREARRAYARRAY.ARRAYARRAY_BOOL[4][3] := NOT RETAINTEST_AUTO_STRUCTUREARRAYARRAY.ARRAYARRAY_BOOL[4][3];
    RETAINTEST_AUTO_STRUCTUREARRAYARRAY.ARRAYARRAY_BOOL[4][4] := NOT RETAINTEST_AUTO_STRUCTUREARRAYARRAY.ARRAYARRAY_BOOL[4][4];
    RETAINTEST_AUTO_STRUCTUREARRAYARRAY.ARRAYARRAY_BOOL[4][5] := NOT RETAINTEST_AUTO_STRUCTUREARRAYARRAY.ARRAYARRAY_BOOL[4][5];
    RETAINTEST_AUTO_STRUCTUREARRAYARRAY.ARRAYARRAY_BOOL[4][6] := NOT RETAINTEST_AUTO_STRUCTUREARRAYARRAY.ARRAYARRAY_BOOL[4][6];
    RETAINTEST_AUTO_STRUCTUREARRAYARRAY.ARRAYARRAY_BOOL[4][7] := NOT RETAINTEST_AUTO_STRUCTUREARRAYARRAY.ARRAYARRAY_BOOL[4][7];
    RETAINTEST_AUTO_STRUCTUREARRAYARRAY.ARRAYARRAY_BOOL[4][8] := NOT RETAINTEST_AUTO_STRUCTUREARRAYARRAY.ARRAYARRAY_BOOL[4][8];
    RETAINTEST_AUTO_STRUCTUREARRAYARRAY.ARRAYARRAY_BOOL[4][9] := NOT RETAINTEST_AUTO_STRUCTUREARRAYARRAY.ARRAYARRAY_BOOL[4][9];

    RETAINTEST_AUTO_STRUCTUREARRAYARRAY.ARRAYARRAY_BOOL[5][0] := NOT RETAINTEST_AUTO_STRUCTUREARRAYARRAY.ARRAYARRAY_BOOL[5][0];
    RETAINTEST_AUTO_STRUCTUREARRAYARRAY.ARRAYARRAY_BOOL[5][1] := NOT RETAINTEST_AUTO_STRUCTUREARRAYARRAY.ARRAYARRAY_BOOL[5][1];
    RETAINTEST_AUTO_STRUCTUREARRAYARRAY.ARRAYARRAY_BOOL[5][2] := NOT RETAINTEST_AUTO_STRUCTUREARRAYARRAY.ARRAYARRAY_BOOL[5][2];
    RETAINTEST_AUTO_STRUCTUREARRAYARRAY.ARRAYARRAY_BOOL[5][3] := NOT RETAINTEST_AUTO_STRUCTUREARRAYARRAY.ARRAYARRAY_BOOL[5][3];
    RETAINTEST_AUTO_STRUCTUREARRAYARRAY.ARRAYARRAY_BOOL[5][4] := NOT RETAINTEST_AUTO_STRUCTUREARRAYARRAY.ARRAYARRAY_BOOL[5][4];
    RETAINTEST_AUTO_STRUCTUREARRAYARRAY.ARRAYARRAY_BOOL[5][5] := NOT RETAINTEST_AUTO_STRUCTUREARRAYARRAY.ARRAYARRAY_BOOL[5][5];
    RETAINTEST_AUTO_STRUCTUREARRAYARRAY.ARRAYARRAY_BOOL[5][6] := NOT RETAINTEST_AUTO_STRUCTUREARRAYARRAY.ARRAYARRAY_BOOL[5][6];
    RETAINTEST_AUTO_STRUCTUREARRAYARRAY.ARRAYARRAY_BOOL[5][7] := NOT RETAINTEST_AUTO_STRUCTUREARRAYARRAY.ARRAYARRAY_BOOL[5][7];
    RETAINTEST_AUTO_STRUCTUREARRAYARRAY.ARRAYARRAY_BOOL[5][8] := NOT RETAINTEST_AUTO_STRUCTUREARRAYARRAY.ARRAYARRAY_BOOL[5][8];
    RETAINTEST_AUTO_STRUCTUREARRAYARRAY.ARRAYARRAY_BOOL[5][9] := NOT RETAINTEST_AUTO_STRUCTUREARRAYARRAY.ARRAYARRAY_BOOL[5][9];

    RETAINTEST_AUTO_STRUCTUREARRAYARRAY.ARRAYARRAY_BOOL[6][0] := NOT RETAINTEST_AUTO_STRUCTUREARRAYARRAY.ARRAYARRAY_BOOL[6][0];
    RETAINTEST_AUTO_STRUCTUREARRAYARRAY.ARRAYARRAY_BOOL[6][1] := NOT RETAINTEST_AUTO_STRUCTUREARRAYARRAY.ARRAYARRAY_BOOL[6][1];
    RETAINTEST_AUTO_STRUCTUREARRAYARRAY.ARRAYARRAY_BOOL[6][2] := NOT RETAINTEST_AUTO_STRUCTUREARRAYARRAY.ARRAYARRAY_BOOL[6][2];
    RETAINTEST_AUTO_STRUCTUREARRAYARRAY.ARRAYARRAY_BOOL[6][3] := NOT RETAINTEST_AUTO_STRUCTUREARRAYARRAY.ARRAYARRAY_BOOL[6][3];
    RETAINTEST_AUTO_STRUCTUREARRAYARRAY.ARRAYARRAY_BOOL[6][4] := NOT RETAINTEST_AUTO_STRUCTUREARRAYARRAY.ARRAYARRAY_BOOL[6][4];
    RETAINTEST_AUTO_STRUCTUREARRAYARRAY.ARRAYARRAY_BOOL[6][5] := NOT RETAINTEST_AUTO_STRUCTUREARRAYARRAY.ARRAYARRAY_BOOL[6][5];
    RETAINTEST_AUTO_STRUCTUREARRAYARRAY.ARRAYARRAY_BOOL[6][6] := NOT RETAINTEST_AUTO_STRUCTUREARRAYARRAY.ARRAYARRAY_BOOL[6][6];
    RETAINTEST_AUTO_STRUCTUREARRAYARRAY.ARRAYARRAY_BOOL[6][7] := NOT RETAINTEST_AUTO_STRUCTUREARRAYARRAY.ARRAYARRAY_BOOL[6][7];
    RETAINTEST_AUTO_STRUCTUREARRAYARRAY.ARRAYARRAY_BOOL[6][8] := NOT RETAINTEST_AUTO_STRUCTUREARRAYARRAY.ARRAYARRAY_BOOL[6][8];
    RETAINTEST_AUTO_STRUCTUREARRAYARRAY.ARRAYARRAY_BOOL[6][9] := NOT RETAINTEST_AUTO_STRUCTUREARRAYARRAY.ARRAYARRAY_BOOL[6][9];

    RETAINTEST_AUTO_STRUCTUREARRAYARRAY.ARRAYARRAY_BOOL[7][0] := RETAINTEST_AUTO_STRUCTUREARRAYARRAY.ARRAYARRAY_BOOL[6][0];
    RETAINTEST_AUTO_STRUCTUREARRAYARRAY.ARRAYARRAY_BOOL[7][1] := RETAINTEST_AUTO_STRUCTUREARRAYARRAY.ARRAYARRAY_BOOL[6][1];
    RETAINTEST_AUTO_STRUCTUREARRAYARRAY.ARRAYARRAY_BOOL[7][2] := RETAINTEST_AUTO_STRUCTUREARRAYARRAY.ARRAYARRAY_BOOL[6][2];
    RETAINTEST_AUTO_STRUCTUREARRAYARRAY.ARRAYARRAY_BOOL[7][3] := RETAINTEST_AUTO_STRUCTUREARRAYARRAY.ARRAYARRAY_BOOL[6][3];
    RETAINTEST_AUTO_STRUCTUREARRAYARRAY.ARRAYARRAY_BOOL[7][4] := RETAINTEST_AUTO_STRUCTUREARRAYARRAY.ARRAYARRAY_BOOL[6][4];
    RETAINTEST_AUTO_STRUCTUREARRAYARRAY.ARRAYARRAY_BOOL[7][5] := RETAINTEST_AUTO_STRUCTUREARRAYARRAY.ARRAYARRAY_BOOL[6][5];
    RETAINTEST_AUTO_STRUCTUREARRAYARRAY.ARRAYARRAY_BOOL[7][6] := RETAINTEST_AUTO_STRUCTUREARRAYARRAY.ARRAYARRAY_BOOL[6][6];
    RETAINTEST_AUTO_STRUCTUREARRAYARRAY.ARRAYARRAY_BOOL[7][7] := RETAINTEST_AUTO_STRUCTUREARRAYARRAY.ARRAYARRAY_BOOL[6][7];
    RETAINTEST_AUTO_STRUCTUREARRAYARRAY.ARRAYARRAY_BOOL[7][8] := RETAINTEST_AUTO_STRUCTUREARRAYARRAY.ARRAYARRAY_BOOL[6][8];
    RETAINTEST_AUTO_STRUCTUREARRAYARRAY.ARRAYARRAY_BOOL[7][9] := RETAINTEST_AUTO_STRUCTUREARRAYARRAY.ARRAYARRAY_BOOL[6][9];

    RETAINTEST_AUTO_STRUCTUREARRAYARRAY.ARRAYARRAY_BYTE[0][0] := RETAINTEST_AUTO_STRUCTUREARRAYARRAY.ARRAYARRAY_BYTE[0][0] + 1;
    RETAINTEST_AUTO_STRUCTUREARRAYARRAY.ARRAYARRAY_BYTE[0][1] := RETAINTEST_AUTO_STRUCTUREARRAYARRAY.ARRAYARRAY_BYTE[0][1] + 1;
    RETAINTEST_AUTO_STRUCTUREARRAYARRAY.ARRAYARRAY_BYTE[0][2] := RETAINTEST_AUTO_STRUCTUREARRAYARRAY.ARRAYARRAY_BYTE[0][2] + 1;
    RETAINTEST_AUTO_STRUCTUREARRAYARRAY.ARRAYARRAY_BYTE[0][3] := RETAINTEST_AUTO_STRUCTUREARRAYARRAY.ARRAYARRAY_BYTE[0][3] + 1;
    RETAINTEST_AUTO_STRUCTUREARRAYARRAY.ARRAYARRAY_BYTE[0][4] := RETAINTEST_AUTO_STRUCTUREARRAYARRAY.ARRAYARRAY_BYTE[0][4] + 1;
    RETAINTEST_AUTO_STRUCTUREARRAYARRAY.ARRAYARRAY_BYTE[0][5] := RETAINTEST_AUTO_STRUCTUREARRAYARRAY.ARRAYARRAY_BYTE[0][5] + 1;
    RETAINTEST_AUTO_STRUCTUREARRAYARRAY.ARRAYARRAY_BYTE[0][6] := RETAINTEST_AUTO_STRUCTUREARRAYARRAY.ARRAYARRAY_BYTE[0][6] + 1;
    RETAINTEST_AUTO_STRUCTUREARRAYARRAY.ARRAYARRAY_BYTE[0][7] := RETAINTEST_AUTO_STRUCTUREARRAYARRAY.ARRAYARRAY_BYTE[0][7] + 1;
    RETAINTEST_AUTO_STRUCTUREARRAYARRAY.ARRAYARRAY_BYTE[0][8] := RETAINTEST_AUTO_STRUCTUREARRAYARRAY.ARRAYARRAY_BYTE[0][6];
    RETAINTEST_AUTO_STRUCTUREARRAYARRAY.ARRAYARRAY_BYTE[0][9] := RETAINTEST_AUTO_STRUCTUREARRAYARRAY.ARRAYARRAY_BYTE[0][7];

    RETAINTEST_AUTO_STRUCTUREARRAYARRAY.ARRAYARRAY_BYTE[1][0] := RETAINTEST_AUTO_STRUCTUREARRAYARRAY.ARRAYARRAY_BYTE[1][0] + 1;
    RETAINTEST_AUTO_STRUCTUREARRAYARRAY.ARRAYARRAY_BYTE[1][1] := RETAINTEST_AUTO_STRUCTUREARRAYARRAY.ARRAYARRAY_BYTE[1][1] + 1;
    RETAINTEST_AUTO_STRUCTUREARRAYARRAY.ARRAYARRAY_BYTE[1][2] := RETAINTEST_AUTO_STRUCTUREARRAYARRAY.ARRAYARRAY_BYTE[1][2] + 1;
    RETAINTEST_AUTO_STRUCTUREARRAYARRAY.ARRAYARRAY_BYTE[1][3] := RETAINTEST_AUTO_STRUCTUREARRAYARRAY.ARRAYARRAY_BYTE[1][3] + 1;
    RETAINTEST_AUTO_STRUCTUREARRAYARRAY.ARRAYARRAY_BYTE[1][4] := RETAINTEST_AUTO_STRUCTUREARRAYARRAY.ARRAYARRAY_BYTE[1][4] + 1;
    RETAINTEST_AUTO_STRUCTUREARRAYARRAY.ARRAYARRAY_BYTE[1][5] := RETAINTEST_AUTO_STRUCTUREARRAYARRAY.ARRAYARRAY_BYTE[1][5] + 1;
    RETAINTEST_AUTO_STRUCTUREARRAYARRAY.ARRAYARRAY_BYTE[1][6] := RETAINTEST_AUTO_STRUCTUREARRAYARRAY.ARRAYARRAY_BYTE[1][6] + 1;
    RETAINTEST_AUTO_STRUCTUREARRAYARRAY.ARRAYARRAY_BYTE[1][7] := RETAINTEST_AUTO_STRUCTUREARRAYARRAY.ARRAYARRAY_BYTE[1][7] + 1;
    RETAINTEST_AUTO_STRUCTUREARRAYARRAY.ARRAYARRAY_BYTE[1][8] := RETAINTEST_AUTO_STRUCTUREARRAYARRAY.ARRAYARRAY_BYTE[1][6];
    RETAINTEST_AUTO_STRUCTUREARRAYARRAY.ARRAYARRAY_BYTE[1][9] := RETAINTEST_AUTO_STRUCTUREARRAYARRAY.ARRAYARRAY_BYTE[1][7];

    RETAINTEST_AUTO_STRUCTUREARRAYARRAY.ARRAYARRAY_BYTE[2][0] := RETAINTEST_AUTO_STRUCTUREARRAYARRAY.ARRAYARRAY_BYTE[2][0] + 1;
    RETAINTEST_AUTO_STRUCTUREARRAYARRAY.ARRAYARRAY_BYTE[2][1] := RETAINTEST_AUTO_STRUCTUREARRAYARRAY.ARRAYARRAY_BYTE[2][1] + 1;
    RETAINTEST_AUTO_STRUCTUREARRAYARRAY.ARRAYARRAY_BYTE[2][2] := RETAINTEST_AUTO_STRUCTUREARRAYARRAY.ARRAYARRAY_BYTE[2][2] + 1;
    RETAINTEST_AUTO_STRUCTUREARRAYARRAY.ARRAYARRAY_BYTE[2][3] := RETAINTEST_AUTO_STRUCTUREARRAYARRAY.ARRAYARRAY_BYTE[2][3] + 1;
    RETAINTEST_AUTO_STRUCTUREARRAYARRAY.ARRAYARRAY_BYTE[2][4] := RETAINTEST_AUTO_STRUCTUREARRAYARRAY.ARRAYARRAY_BYTE[2][4] + 1;
    RETAINTEST_AUTO_STRUCTUREARRAYARRAY.ARRAYARRAY_BYTE[2][5] := RETAINTEST_AUTO_STRUCTUREARRAYARRAY.ARRAYARRAY_BYTE[2][5] + 1;
    RETAINTEST_AUTO_STRUCTUREARRAYARRAY.ARRAYARRAY_BYTE[2][6] := RETAINTEST_AUTO_STRUCTUREARRAYARRAY.ARRAYARRAY_BYTE[2][6] + 1;
    RETAINTEST_AUTO_STRUCTUREARRAYARRAY.ARRAYARRAY_BYTE[2][7] := RETAINTEST_AUTO_STRUCTUREARRAYARRAY.ARRAYARRAY_BYTE[2][7] + 1;
    RETAINTEST_AUTO_STRUCTUREARRAYARRAY.ARRAYARRAY_BYTE[2][8] := RETAINTEST_AUTO_STRUCTUREARRAYARRAY.ARRAYARRAY_BYTE[2][8] + 1;
    RETAINTEST_AUTO_STRUCTUREARRAYARRAY.ARRAYARRAY_BYTE[2][9] := RETAINTEST_AUTO_STRUCTUREARRAYARRAY.ARRAYARRAY_BYTE[2][9] + 1;

    RETAINTEST_AUTO_STRUCTUREARRAYARRAY.ARRAYARRAY_BYTE[3][0] := RETAINTEST_AUTO_STRUCTUREARRAYARRAY.ARRAYARRAY_BYTE[3][0] + 1;
    RETAINTEST_AUTO_STRUCTUREARRAYARRAY.ARRAYARRAY_BYTE[3][1] := RETAINTEST_AUTO_STRUCTUREARRAYARRAY.ARRAYARRAY_BYTE[3][1] + 1;
    RETAINTEST_AUTO_STRUCTUREARRAYARRAY.ARRAYARRAY_BYTE[3][2] := RETAINTEST_AUTO_STRUCTUREARRAYARRAY.ARRAYARRAY_BYTE[3][2] + 1;
    RETAINTEST_AUTO_STRUCTUREARRAYARRAY.ARRAYARRAY_BYTE[3][3] := RETAINTEST_AUTO_STRUCTUREARRAYARRAY.ARRAYARRAY_BYTE[3][3] + 1;
    RETAINTEST_AUTO_STRUCTUREARRAYARRAY.ARRAYARRAY_BYTE[3][4] := RETAINTEST_AUTO_STRUCTUREARRAYARRAY.ARRAYARRAY_BYTE[3][4] + 1;
    RETAINTEST_AUTO_STRUCTUREARRAYARRAY.ARRAYARRAY_BYTE[3][5] := RETAINTEST_AUTO_STRUCTUREARRAYARRAY.ARRAYARRAY_BYTE[3][5] + 1;
    RETAINTEST_AUTO_STRUCTUREARRAYARRAY.ARRAYARRAY_BYTE[3][6] := RETAINTEST_AUTO_STRUCTUREARRAYARRAY.ARRAYARRAY_BYTE[3][6] + 1;
    RETAINTEST_AUTO_STRUCTUREARRAYARRAY.ARRAYARRAY_BYTE[3][7] := RETAINTEST_AUTO_STRUCTUREARRAYARRAY.ARRAYARRAY_BYTE[3][7] + 1;
    RETAINTEST_AUTO_STRUCTUREARRAYARRAY.ARRAYARRAY_BYTE[3][8] := RETAINTEST_AUTO_STRUCTUREARRAYARRAY.ARRAYARRAY_BYTE[3][8] + 1;
    RETAINTEST_AUTO_STRUCTUREARRAYARRAY.ARRAYARRAY_BYTE[3][9] := RETAINTEST_AUTO_STRUCTUREARRAYARRAY.ARRAYARRAY_BYTE[3][9] + 1;

    RETAINTEST_AUTO_STRUCTUREARRAYARRAY.ARRAYARRAY_BYTE[4][0] := RETAINTEST_AUTO_STRUCTUREARRAYARRAY.ARRAYARRAY_BYTE[4][0] + 1;
    RETAINTEST_AUTO_STRUCTUREARRAYARRAY.ARRAYARRAY_BYTE[4][1] := RETAINTEST_AUTO_STRUCTUREARRAYARRAY.ARRAYARRAY_BYTE[4][1] + 1;
    RETAINTEST_AUTO_STRUCTUREARRAYARRAY.ARRAYARRAY_BYTE[4][2] := RETAINTEST_AUTO_STRUCTUREARRAYARRAY.ARRAYARRAY_BYTE[4][2] + 1;
    RETAINTEST_AUTO_STRUCTUREARRAYARRAY.ARRAYARRAY_BYTE[4][3] := RETAINTEST_AUTO_STRUCTUREARRAYARRAY.ARRAYARRAY_BYTE[4][3] + 1;
    RETAINTEST_AUTO_STRUCTUREARRAYARRAY.ARRAYARRAY_BYTE[4][4] := RETAINTEST_AUTO_STRUCTUREARRAYARRAY.ARRAYARRAY_BYTE[4][4] + 1;
    RETAINTEST_AUTO_STRUCTUREARRAYARRAY.ARRAYARRAY_BYTE[4][5] := RETAINTEST_AUTO_STRUCTUREARRAYARRAY.ARRAYARRAY_BYTE[4][5] + 1;
    RETAINTEST_AUTO_STRUCTUREARRAYARRAY.ARRAYARRAY_BYTE[4][6] := RETAINTEST_AUTO_STRUCTUREARRAYARRAY.ARRAYARRAY_BYTE[4][6] + 1;
    RETAINTEST_AUTO_STRUCTUREARRAYARRAY.ARRAYARRAY_BYTE[4][7] := RETAINTEST_AUTO_STRUCTUREARRAYARRAY.ARRAYARRAY_BYTE[4][7] + 1;
    RETAINTEST_AUTO_STRUCTUREARRAYARRAY.ARRAYARRAY_BYTE[4][8] := RETAINTEST_AUTO_STRUCTUREARRAYARRAY.ARRAYARRAY_BYTE[4][8] + 1;
    RETAINTEST_AUTO_STRUCTUREARRAYARRAY.ARRAYARRAY_BYTE[4][9] := RETAINTEST_AUTO_STRUCTUREARRAYARRAY.ARRAYARRAY_BYTE[4][9] + 1;

    RETAINTEST_AUTO_STRUCTUREARRAYARRAY.ARRAYARRAY_BYTE[5][0] := RETAINTEST_AUTO_STRUCTUREARRAYARRAY.ARRAYARRAY_BYTE[5][0] + 1;
    RETAINTEST_AUTO_STRUCTUREARRAYARRAY.ARRAYARRAY_BYTE[5][1] := RETAINTEST_AUTO_STRUCTUREARRAYARRAY.ARRAYARRAY_BYTE[5][1] + 1;
    RETAINTEST_AUTO_STRUCTUREARRAYARRAY.ARRAYARRAY_BYTE[5][2] := RETAINTEST_AUTO_STRUCTUREARRAYARRAY.ARRAYARRAY_BYTE[5][2] + 1;
    RETAINTEST_AUTO_STRUCTUREARRAYARRAY.ARRAYARRAY_BYTE[5][3] := RETAINTEST_AUTO_STRUCTUREARRAYARRAY.ARRAYARRAY_BYTE[5][3] + 1;
    RETAINTEST_AUTO_STRUCTUREARRAYARRAY.ARRAYARRAY_BYTE[5][4] := RETAINTEST_AUTO_STRUCTUREARRAYARRAY.ARRAYARRAY_BYTE[5][4] + 1;
    RETAINTEST_AUTO_STRUCTUREARRAYARRAY.ARRAYARRAY_BYTE[5][5] := RETAINTEST_AUTO_STRUCTUREARRAYARRAY.ARRAYARRAY_BYTE[5][5] + 1;
    RETAINTEST_AUTO_STRUCTUREARRAYARRAY.ARRAYARRAY_BYTE[5][6] := RETAINTEST_AUTO_STRUCTUREARRAYARRAY.ARRAYARRAY_BYTE[5][6] + 1;
    RETAINTEST_AUTO_STRUCTUREARRAYARRAY.ARRAYARRAY_BYTE[5][7] := RETAINTEST_AUTO_STRUCTUREARRAYARRAY.ARRAYARRAY_BYTE[5][7] + 1;
    RETAINTEST_AUTO_STRUCTUREARRAYARRAY.ARRAYARRAY_BYTE[5][8] := RETAINTEST_AUTO_STRUCTUREARRAYARRAY.ARRAYARRAY_BYTE[5][8] + 1;
    RETAINTEST_AUTO_STRUCTUREARRAYARRAY.ARRAYARRAY_BYTE[5][9] := RETAINTEST_AUTO_STRUCTUREARRAYARRAY.ARRAYARRAY_BYTE[5][9] + 1;

    RETAINTEST_AUTO_STRUCTUREARRAYARRAY.ARRAYARRAY_BYTE[6][0] := RETAINTEST_AUTO_STRUCTUREARRAYARRAY.ARRAYARRAY_BYTE[6][0] + 1;
    RETAINTEST_AUTO_STRUCTUREARRAYARRAY.ARRAYARRAY_BYTE[6][1] := RETAINTEST_AUTO_STRUCTUREARRAYARRAY.ARRAYARRAY_BYTE[6][1] + 1;
    RETAINTEST_AUTO_STRUCTUREARRAYARRAY.ARRAYARRAY_BYTE[6][2] := RETAINTEST_AUTO_STRUCTUREARRAYARRAY.ARRAYARRAY_BYTE[6][2] + 1;
    RETAINTEST_AUTO_STRUCTUREARRAYARRAY.ARRAYARRAY_BYTE[6][3] := RETAINTEST_AUTO_STRUCTUREARRAYARRAY.ARRAYARRAY_BYTE[6][3] + 1;
    RETAINTEST_AUTO_STRUCTUREARRAYARRAY.ARRAYARRAY_BYTE[6][4] := RETAINTEST_AUTO_STRUCTUREARRAYARRAY.ARRAYARRAY_BYTE[6][4] + 1;
    RETAINTEST_AUTO_STRUCTUREARRAYARRAY.ARRAYARRAY_BYTE[6][5] := RETAINTEST_AUTO_STRUCTUREARRAYARRAY.ARRAYARRAY_BYTE[6][5] + 1;
    RETAINTEST_AUTO_STRUCTUREARRAYARRAY.ARRAYARRAY_BYTE[6][6] := RETAINTEST_AUTO_STRUCTUREARRAYARRAY.ARRAYARRAY_BYTE[6][6] + 1;
    RETAINTEST_AUTO_STRUCTUREARRAYARRAY.ARRAYARRAY_BYTE[6][7] := RETAINTEST_AUTO_STRUCTUREARRAYARRAY.ARRAYARRAY_BYTE[6][7] + 1;
    RETAINTEST_AUTO_STRUCTUREARRAYARRAY.ARRAYARRAY_BYTE[6][8] := RETAINTEST_AUTO_STRUCTUREARRAYARRAY.ARRAYARRAY_BYTE[6][8] + 1;
    RETAINTEST_AUTO_STRUCTUREARRAYARRAY.ARRAYARRAY_BYTE[6][9] := RETAINTEST_AUTO_STRUCTUREARRAYARRAY.ARRAYARRAY_BYTE[6][9] + 1;

    RETAINTEST_AUTO_STRUCTUREARRAYARRAY.ARRAYARRAY_BYTE[7][0] := RETAINTEST_AUTO_STRUCTUREARRAYARRAY.ARRAYARRAY_BYTE[6][0];
    RETAINTEST_AUTO_STRUCTUREARRAYARRAY.ARRAYARRAY_BYTE[7][1] := RETAINTEST_AUTO_STRUCTUREARRAYARRAY.ARRAYARRAY_BYTE[6][1];
    RETAINTEST_AUTO_STRUCTUREARRAYARRAY.ARRAYARRAY_BYTE[7][2] := RETAINTEST_AUTO_STRUCTUREARRAYARRAY.ARRAYARRAY_BYTE[6][2];
    RETAINTEST_AUTO_STRUCTUREARRAYARRAY.ARRAYARRAY_BYTE[7][3] := RETAINTEST_AUTO_STRUCTUREARRAYARRAY.ARRAYARRAY_BYTE[6][3];
    RETAINTEST_AUTO_STRUCTUREARRAYARRAY.ARRAYARRAY_BYTE[7][4] := RETAINTEST_AUTO_STRUCTUREARRAYARRAY.ARRAYARRAY_BYTE[6][4];
    RETAINTEST_AUTO_STRUCTUREARRAYARRAY.ARRAYARRAY_BYTE[7][5] := RETAINTEST_AUTO_STRUCTUREARRAYARRAY.ARRAYARRAY_BYTE[6][5];
    RETAINTEST_AUTO_STRUCTUREARRAYARRAY.ARRAYARRAY_BYTE[7][6] := RETAINTEST_AUTO_STRUCTUREARRAYARRAY.ARRAYARRAY_BYTE[6][6];
    RETAINTEST_AUTO_STRUCTUREARRAYARRAY.ARRAYARRAY_BYTE[7][7] := RETAINTEST_AUTO_STRUCTUREARRAYARRAY.ARRAYARRAY_BYTE[6][7];
    RETAINTEST_AUTO_STRUCTUREARRAYARRAY.ARRAYARRAY_BYTE[7][8] := RETAINTEST_AUTO_STRUCTUREARRAYARRAY.ARRAYARRAY_BYTE[6][8];
    RETAINTEST_AUTO_STRUCTUREARRAYARRAY.ARRAYARRAY_BYTE[7][9] := RETAINTEST_AUTO_STRUCTUREARRAYARRAY.ARRAYARRAY_BYTE[6][9];

    RETAINTEST_AUTO_STRUCTUREARRAYARRAY.ARRAYARRAY_DATE[0][0] := ANY_TO_DATE(1445385600 + RETAINTEST_AUTO_STRUCTUREARRAYARRAY.ARRAYARRAY_DINT[0][0] * 86400);
    RETAINTEST_AUTO_STRUCTUREARRAYARRAY.ARRAYARRAY_DATE[0][1] := ANY_TO_DATE(1445385600 + RETAINTEST_AUTO_STRUCTUREARRAYARRAY.ARRAYARRAY_DINT[0][1] * 86400);
    RETAINTEST_AUTO_STRUCTUREARRAYARRAY.ARRAYARRAY_DATE[0][2] := ANY_TO_DATE(1445385600 + RETAINTEST_AUTO_STRUCTUREARRAYARRAY.ARRAYARRAY_DINT[0][2] * 86400);
    RETAINTEST_AUTO_STRUCTUREARRAYARRAY.ARRAYARRAY_DATE[0][3] := ANY_TO_DATE(1445385600 + RETAINTEST_AUTO_STRUCTUREARRAYARRAY.ARRAYARRAY_DINT[0][3] * 86400);
    RETAINTEST_AUTO_STRUCTUREARRAYARRAY.ARRAYARRAY_DATE[0][4] := ANY_TO_DATE(1445385600 + RETAINTEST_AUTO_STRUCTUREARRAYARRAY.ARRAYARRAY_DINT[0][4] * 86400);
    RETAINTEST_AUTO_STRUCTUREARRAYARRAY.ARRAYARRAY_DATE[0][5] := ANY_TO_DATE(1445385600 + RETAINTEST_AUTO_STRUCTUREARRAYARRAY.ARRAYARRAY_DINT[0][5] * 86400);
    RETAINTEST_AUTO_STRUCTUREARRAYARRAY.ARRAYARRAY_DATE[0][6] := ANY_TO_DATE(1445385600 + RETAINTEST_AUTO_STRUCTUREARRAYARRAY.ARRAYARRAY_DINT[0][6] * 86400);
    RETAINTEST_AUTO_STRUCTUREARRAYARRAY.ARRAYARRAY_DATE[0][7] := ANY_TO_DATE(1445385600 + RETAINTEST_AUTO_STRUCTUREARRAYARRAY.ARRAYARRAY_DINT[0][7] * 86400);
    RETAINTEST_AUTO_STRUCTUREARRAYARRAY.ARRAYARRAY_DATE[0][8] := RETAINTEST_AUTO_STRUCTUREARRAYARRAY.ARRAYARRAY_DATE[0][6];
    RETAINTEST_AUTO_STRUCTUREARRAYARRAY.ARRAYARRAY_DATE[0][9] := RETAINTEST_AUTO_STRUCTUREARRAYARRAY.ARRAYARRAY_DATE[0][7];

    RETAINTEST_AUTO_STRUCTUREARRAYARRAY.ARRAYARRAY_DATE[1][0] := ANY_TO_DATE(1445385600 + RETAINTEST_AUTO_STRUCTUREARRAYARRAY.ARRAYARRAY_DINT[1][0] * 86400);
    RETAINTEST_AUTO_STRUCTUREARRAYARRAY.ARRAYARRAY_DATE[1][1] := ANY_TO_DATE(1445385600 + RETAINTEST_AUTO_STRUCTUREARRAYARRAY.ARRAYARRAY_DINT[1][1] * 86400);
    RETAINTEST_AUTO_STRUCTUREARRAYARRAY.ARRAYARRAY_DATE[1][2] := ANY_TO_DATE(1445385600 + RETAINTEST_AUTO_STRUCTUREARRAYARRAY.ARRAYARRAY_DINT[1][2] * 86400);
    RETAINTEST_AUTO_STRUCTUREARRAYARRAY.ARRAYARRAY_DATE[1][3] := ANY_TO_DATE(1445385600 + RETAINTEST_AUTO_STRUCTUREARRAYARRAY.ARRAYARRAY_DINT[1][3] * 86400);
    RETAINTEST_AUTO_STRUCTUREARRAYARRAY.ARRAYARRAY_DATE[1][4] := ANY_TO_DATE(1445385600 + RETAINTEST_AUTO_STRUCTUREARRAYARRAY.ARRAYARRAY_DINT[1][4] * 86400);
    RETAINTEST_AUTO_STRUCTUREARRAYARRAY.ARRAYARRAY_DATE[1][5] := ANY_TO_DATE(1445385600 + RETAINTEST_AUTO_STRUCTUREARRAYARRAY.ARRAYARRAY_DINT[1][5] * 86400);
    RETAINTEST_AUTO_STRUCTUREARRAYARRAY.ARRAYARRAY_DATE[1][6] := ANY_TO_DATE(1445385600 + RETAINTEST_AUTO_STRUCTUREARRAYARRAY.ARRAYARRAY_DINT[1][6] * 86400);
    RETAINTEST_AUTO_STRUCTUREARRAYARRAY.ARRAYARRAY_DATE[1][7] := ANY_TO_DATE(1445385600 + RETAINTEST_AUTO_STRUCTUREARRAYARRAY.ARRAYARRAY_DINT[1][7] * 86400);
    RETAINTEST_AUTO_STRUCTUREARRAYARRAY.ARRAYARRAY_DATE[1][8] := RETAINTEST_AUTO_STRUCTUREARRAYARRAY.ARRAYARRAY_DATE[1][6];
    RETAINTEST_AUTO_STRUCTUREARRAYARRAY.ARRAYARRAY_DATE[1][9] := RETAINTEST_AUTO_STRUCTUREARRAYARRAY.ARRAYARRAY_DATE[1][7];

    RETAINTEST_AUTO_STRUCTUREARRAYARRAY.ARRAYARRAY_DATE[2][0] := ANY_TO_DATE(1445385600 + RETAINTEST_AUTO_STRUCTUREARRAYARRAY.ARRAYARRAY_DINT[2][0] * 86400);
    RETAINTEST_AUTO_STRUCTUREARRAYARRAY.ARRAYARRAY_DATE[2][1] := ANY_TO_DATE(1445385600 + RETAINTEST_AUTO_STRUCTUREARRAYARRAY.ARRAYARRAY_DINT[2][1] * 86400);
    RETAINTEST_AUTO_STRUCTUREARRAYARRAY.ARRAYARRAY_DATE[2][2] := ANY_TO_DATE(1445385600 + RETAINTEST_AUTO_STRUCTUREARRAYARRAY.ARRAYARRAY_DINT[2][2] * 86400);
    RETAINTEST_AUTO_STRUCTUREARRAYARRAY.ARRAYARRAY_DATE[2][3] := ANY_TO_DATE(1445385600 + RETAINTEST_AUTO_STRUCTUREARRAYARRAY.ARRAYARRAY_DINT[2][3] * 86400);
    RETAINTEST_AUTO_STRUCTUREARRAYARRAY.ARRAYARRAY_DATE[2][4] := ANY_TO_DATE(1445385600 + RETAINTEST_AUTO_STRUCTUREARRAYARRAY.ARRAYARRAY_DINT[2][4] * 86400);
    RETAINTEST_AUTO_STRUCTUREARRAYARRAY.ARRAYARRAY_DATE[2][5] := ANY_TO_DATE(1445385600 + RETAINTEST_AUTO_STRUCTUREARRAYARRAY.ARRAYARRAY_DINT[2][5] * 86400);
    RETAINTEST_AUTO_STRUCTUREARRAYARRAY.ARRAYARRAY_DATE[2][6] := ANY_TO_DATE(1445385600 + RETAINTEST_AUTO_STRUCTUREARRAYARRAY.ARRAYARRAY_DINT[2][6] * 86400);
    RETAINTEST_AUTO_STRUCTUREARRAYARRAY.ARRAYARRAY_DATE[2][7] := ANY_TO_DATE(1445385600 + RETAINTEST_AUTO_STRUCTUREARRAYARRAY.ARRAYARRAY_DINT[2][7] * 86400);
    RETAINTEST_AUTO_STRUCTUREARRAYARRAY.ARRAYARRAY_DATE[2][8] := ANY_TO_DATE(1445385600 + RETAINTEST_AUTO_STRUCTUREARRAYARRAY.ARRAYARRAY_DINT[2][8] * 86400);
    RETAINTEST_AUTO_STRUCTUREARRAYARRAY.ARRAYARRAY_DATE[2][9] := ANY_TO_DATE(1445385600 + RETAINTEST_AUTO_STRUCTUREARRAYARRAY.ARRAYARRAY_DINT[2][9] * 86400);

    RETAINTEST_AUTO_STRUCTUREARRAYARRAY.ARRAYARRAY_DATE[3][0] := ANY_TO_DATE(1445385600 + RETAINTEST_AUTO_STRUCTUREARRAYARRAY.ARRAYARRAY_DINT[3][0] * 86400);
    RETAINTEST_AUTO_STRUCTUREARRAYARRAY.ARRAYARRAY_DATE[3][1] := ANY_TO_DATE(1445385600 + RETAINTEST_AUTO_STRUCTUREARRAYARRAY.ARRAYARRAY_DINT[3][1] * 86400);
    RETAINTEST_AUTO_STRUCTUREARRAYARRAY.ARRAYARRAY_DATE[3][2] := ANY_TO_DATE(1445385600 + RETAINTEST_AUTO_STRUCTUREARRAYARRAY.ARRAYARRAY_DINT[3][2] * 86400);
    RETAINTEST_AUTO_STRUCTUREARRAYARRAY.ARRAYARRAY_DATE[3][3] := ANY_TO_DATE(1445385600 + RETAINTEST_AUTO_STRUCTUREARRAYARRAY.ARRAYARRAY_DINT[3][3] * 86400);
    RETAINTEST_AUTO_STRUCTUREARRAYARRAY.ARRAYARRAY_DATE[3][4] := ANY_TO_DATE(1445385600 + RETAINTEST_AUTO_STRUCTUREARRAYARRAY.ARRAYARRAY_DINT[3][4] * 86400);
    RETAINTEST_AUTO_STRUCTUREARRAYARRAY.ARRAYARRAY_DATE[3][5] := ANY_TO_DATE(1445385600 + RETAINTEST_AUTO_STRUCTUREARRAYARRAY.ARRAYARRAY_DINT[3][5] * 86400);
    RETAINTEST_AUTO_STRUCTUREARRAYARRAY.ARRAYARRAY_DATE[3][6] := ANY_TO_DATE(1445385600 + RETAINTEST_AUTO_STRUCTUREARRAYARRAY.ARRAYARRAY_DINT[3][6] * 86400);
    RETAINTEST_AUTO_STRUCTUREARRAYARRAY.ARRAYARRAY_DATE[3][7] := ANY_TO_DATE(1445385600 + RETAINTEST_AUTO_STRUCTUREARRAYARRAY.ARRAYARRAY_DINT[3][7] * 86400);
    RETAINTEST_AUTO_STRUCTUREARRAYARRAY.ARRAYARRAY_DATE[3][8] := ANY_TO_DATE(1445385600 + RETAINTEST_AUTO_STRUCTUREARRAYARRAY.ARRAYARRAY_DINT[3][8] * 86400);
    RETAINTEST_AUTO_STRUCTUREARRAYARRAY.ARRAYARRAY_DATE[3][9] := ANY_TO_DATE(1445385600 + RETAINTEST_AUTO_STRUCTUREARRAYARRAY.ARRAYARRAY_DINT[3][9] * 86400);

    RETAINTEST_AUTO_STRUCTUREARRAYARRAY.ARRAYARRAY_DATE[4][0] := ANY_TO_DATE(1445385600 + RETAINTEST_AUTO_STRUCTUREARRAYARRAY.ARRAYARRAY_DINT[4][0] * 86400);
    RETAINTEST_AUTO_STRUCTUREARRAYARRAY.ARRAYARRAY_DATE[4][1] := ANY_TO_DATE(1445385600 + RETAINTEST_AUTO_STRUCTUREARRAYARRAY.ARRAYARRAY_DINT[4][1] * 86400);
    RETAINTEST_AUTO_STRUCTUREARRAYARRAY.ARRAYARRAY_DATE[4][2] := ANY_TO_DATE(1445385600 + RETAINTEST_AUTO_STRUCTUREARRAYARRAY.ARRAYARRAY_DINT[4][2] * 86400);
    RETAINTEST_AUTO_STRUCTUREARRAYARRAY.ARRAYARRAY_DATE[4][3] := ANY_TO_DATE(1445385600 + RETAINTEST_AUTO_STRUCTUREARRAYARRAY.ARRAYARRAY_DINT[4][3] * 86400);
    RETAINTEST_AUTO_STRUCTUREARRAYARRAY.ARRAYARRAY_DATE[4][4] := ANY_TO_DATE(1445385600 + RETAINTEST_AUTO_STRUCTUREARRAYARRAY.ARRAYARRAY_DINT[4][4] * 86400);
    RETAINTEST_AUTO_STRUCTUREARRAYARRAY.ARRAYARRAY_DATE[4][5] := ANY_TO_DATE(1445385600 + RETAINTEST_AUTO_STRUCTUREARRAYARRAY.ARRAYARRAY_DINT[4][5] * 86400);
    RETAINTEST_AUTO_STRUCTUREARRAYARRAY.ARRAYARRAY_DATE[4][6] := ANY_TO_DATE(1445385600 + RETAINTEST_AUTO_STRUCTUREARRAYARRAY.ARRAYARRAY_DINT[4][6] * 86400);
    RETAINTEST_AUTO_STRUCTUREARRAYARRAY.ARRAYARRAY_DATE[4][7] := ANY_TO_DATE(1445385600 + RETAINTEST_AUTO_STRUCTUREARRAYARRAY.ARRAYARRAY_DINT[4][7] * 86400);
    RETAINTEST_AUTO_STRUCTUREARRAYARRAY.ARRAYARRAY_DATE[4][8] := ANY_TO_DATE(1445385600 + RETAINTEST_AUTO_STRUCTUREARRAYARRAY.ARRAYARRAY_DINT[4][8] * 86400);
    RETAINTEST_AUTO_STRUCTUREARRAYARRAY.ARRAYARRAY_DATE[4][9] := ANY_TO_DATE(1445385600 + RETAINTEST_AUTO_STRUCTUREARRAYARRAY.ARRAYARRAY_DINT[4][9] * 86400);

    RETAINTEST_AUTO_STRUCTUREARRAYARRAY.ARRAYARRAY_DATE[5][0] := ANY_TO_DATE(1445385600 + RETAINTEST_AUTO_STRUCTUREARRAYARRAY.ARRAYARRAY_DINT[5][0] * 86400);
    RETAINTEST_AUTO_STRUCTUREARRAYARRAY.ARRAYARRAY_DATE[5][1] := ANY_TO_DATE(1445385600 + RETAINTEST_AUTO_STRUCTUREARRAYARRAY.ARRAYARRAY_DINT[5][1] * 86400);
    RETAINTEST_AUTO_STRUCTUREARRAYARRAY.ARRAYARRAY_DATE[5][2] := ANY_TO_DATE(1445385600 + RETAINTEST_AUTO_STRUCTUREARRAYARRAY.ARRAYARRAY_DINT[5][2] * 86400);
    RETAINTEST_AUTO_STRUCTUREARRAYARRAY.ARRAYARRAY_DATE[5][3] := ANY_TO_DATE(1445385600 + RETAINTEST_AUTO_STRUCTUREARRAYARRAY.ARRAYARRAY_DINT[5][3] * 86400);
    RETAINTEST_AUTO_STRUCTUREARRAYARRAY.ARRAYARRAY_DATE[5][4] := ANY_TO_DATE(1445385600 + RETAINTEST_AUTO_STRUCTUREARRAYARRAY.ARRAYARRAY_DINT[5][4] * 86400);
    RETAINTEST_AUTO_STRUCTUREARRAYARRAY.ARRAYARRAY_DATE[5][5] := ANY_TO_DATE(1445385600 + RETAINTEST_AUTO_STRUCTUREARRAYARRAY.ARRAYARRAY_DINT[5][5] * 86400);
    RETAINTEST_AUTO_STRUCTUREARRAYARRAY.ARRAYARRAY_DATE[5][6] := ANY_TO_DATE(1445385600 + RETAINTEST_AUTO_STRUCTUREARRAYARRAY.ARRAYARRAY_DINT[5][6] * 86400);
    RETAINTEST_AUTO_STRUCTUREARRAYARRAY.ARRAYARRAY_DATE[5][7] := ANY_TO_DATE(1445385600 + RETAINTEST_AUTO_STRUCTUREARRAYARRAY.ARRAYARRAY_DINT[5][7] * 86400);
    RETAINTEST_AUTO_STRUCTUREARRAYARRAY.ARRAYARRAY_DATE[5][8] := ANY_TO_DATE(1445385600 + RETAINTEST_AUTO_STRUCTUREARRAYARRAY.ARRAYARRAY_DINT[5][8] * 86400);
    RETAINTEST_AUTO_STRUCTUREARRAYARRAY.ARRAYARRAY_DATE[5][9] := ANY_TO_DATE(1445385600 + RETAINTEST_AUTO_STRUCTUREARRAYARRAY.ARRAYARRAY_DINT[5][9] * 86400);

    RETAINTEST_AUTO_STRUCTUREARRAYARRAY.ARRAYARRAY_DATE[6][0] := ANY_TO_DATE(1445385600 + RETAINTEST_AUTO_STRUCTUREARRAYARRAY.ARRAYARRAY_DINT[6][0] * 86400);
    RETAINTEST_AUTO_STRUCTUREARRAYARRAY.ARRAYARRAY_DATE[6][1] := ANY_TO_DATE(1445385600 + RETAINTEST_AUTO_STRUCTUREARRAYARRAY.ARRAYARRAY_DINT[6][1] * 86400);
    RETAINTEST_AUTO_STRUCTUREARRAYARRAY.ARRAYARRAY_DATE[6][2] := ANY_TO_DATE(1445385600 + RETAINTEST_AUTO_STRUCTUREARRAYARRAY.ARRAYARRAY_DINT[6][2] * 86400);
    RETAINTEST_AUTO_STRUCTUREARRAYARRAY.ARRAYARRAY_DATE[6][3] := ANY_TO_DATE(1445385600 + RETAINTEST_AUTO_STRUCTUREARRAYARRAY.ARRAYARRAY_DINT[6][3] * 86400);
    RETAINTEST_AUTO_STRUCTUREARRAYARRAY.ARRAYARRAY_DATE[6][4] := ANY_TO_DATE(1445385600 + RETAINTEST_AUTO_STRUCTUREARRAYARRAY.ARRAYARRAY_DINT[6][4] * 86400);
    RETAINTEST_AUTO_STRUCTUREARRAYARRAY.ARRAYARRAY_DATE[6][5] := ANY_TO_DATE(1445385600 + RETAINTEST_AUTO_STRUCTUREARRAYARRAY.ARRAYARRAY_DINT[6][5] * 86400);
    RETAINTEST_AUTO_STRUCTUREARRAYARRAY.ARRAYARRAY_DATE[6][6] := ANY_TO_DATE(1445385600 + RETAINTEST_AUTO_STRUCTUREARRAYARRAY.ARRAYARRAY_DINT[6][6] * 86400);
    RETAINTEST_AUTO_STRUCTUREARRAYARRAY.ARRAYARRAY_DATE[6][7] := ANY_TO_DATE(1445385600 + RETAINTEST_AUTO_STRUCTUREARRAYARRAY.ARRAYARRAY_DINT[6][7] * 86400);
    RETAINTEST_AUTO_STRUCTUREARRAYARRAY.ARRAYARRAY_DATE[6][8] := ANY_TO_DATE(1445385600 + RETAINTEST_AUTO_STRUCTUREARRAYARRAY.ARRAYARRAY_DINT[6][8] * 86400);
    RETAINTEST_AUTO_STRUCTUREARRAYARRAY.ARRAYARRAY_DATE[6][9] := ANY_TO_DATE(1445385600 + RETAINTEST_AUTO_STRUCTUREARRAYARRAY.ARRAYARRAY_DINT[6][9] * 86400);

    RETAINTEST_AUTO_STRUCTUREARRAYARRAY.ARRAYARRAY_DATE[7][0] := RETAINTEST_AUTO_STRUCTUREARRAYARRAY.ARRAYARRAY_DATE[6][0];
    RETAINTEST_AUTO_STRUCTUREARRAYARRAY.ARRAYARRAY_DATE[7][1] := RETAINTEST_AUTO_STRUCTUREARRAYARRAY.ARRAYARRAY_DATE[6][1];
    RETAINTEST_AUTO_STRUCTUREARRAYARRAY.ARRAYARRAY_DATE[7][2] := RETAINTEST_AUTO_STRUCTUREARRAYARRAY.ARRAYARRAY_DATE[6][2];
    RETAINTEST_AUTO_STRUCTUREARRAYARRAY.ARRAYARRAY_DATE[7][3] := RETAINTEST_AUTO_STRUCTUREARRAYARRAY.ARRAYARRAY_DATE[6][3];
    RETAINTEST_AUTO_STRUCTUREARRAYARRAY.ARRAYARRAY_DATE[7][4] := RETAINTEST_AUTO_STRUCTUREARRAYARRAY.ARRAYARRAY_DATE[6][4];
    RETAINTEST_AUTO_STRUCTUREARRAYARRAY.ARRAYARRAY_DATE[7][5] := RETAINTEST_AUTO_STRUCTUREARRAYARRAY.ARRAYARRAY_DATE[6][5];
    RETAINTEST_AUTO_STRUCTUREARRAYARRAY.ARRAYARRAY_DATE[7][6] := RETAINTEST_AUTO_STRUCTUREARRAYARRAY.ARRAYARRAY_DATE[6][6];
    RETAINTEST_AUTO_STRUCTUREARRAYARRAY.ARRAYARRAY_DATE[7][7] := RETAINTEST_AUTO_STRUCTUREARRAYARRAY.ARRAYARRAY_DATE[6][7];
    RETAINTEST_AUTO_STRUCTUREARRAYARRAY.ARRAYARRAY_DATE[7][8] := RETAINTEST_AUTO_STRUCTUREARRAYARRAY.ARRAYARRAY_DATE[6][8];
    RETAINTEST_AUTO_STRUCTUREARRAYARRAY.ARRAYARRAY_DATE[7][9] := RETAINTEST_AUTO_STRUCTUREARRAYARRAY.ARRAYARRAY_DATE[6][9];

    RETAINTEST_AUTO_STRUCTUREARRAYARRAY.ARRAYARRAY_DINT[0][0] := RETAINTEST_AUTO_STRUCTUREARRAYARRAY.ARRAYARRAY_DINT[0][0] + 1;
    RETAINTEST_AUTO_STRUCTUREARRAYARRAY.ARRAYARRAY_DINT[0][1] := RETAINTEST_AUTO_STRUCTUREARRAYARRAY.ARRAYARRAY_DINT[0][1] + 1;
    RETAINTEST_AUTO_STRUCTUREARRAYARRAY.ARRAYARRAY_DINT[0][2] := RETAINTEST_AUTO_STRUCTUREARRAYARRAY.ARRAYARRAY_DINT[0][2] + 1;
    RETAINTEST_AUTO_STRUCTUREARRAYARRAY.ARRAYARRAY_DINT[0][3] := RETAINTEST_AUTO_STRUCTUREARRAYARRAY.ARRAYARRAY_DINT[0][3] + 1;
    RETAINTEST_AUTO_STRUCTUREARRAYARRAY.ARRAYARRAY_DINT[0][4] := RETAINTEST_AUTO_STRUCTUREARRAYARRAY.ARRAYARRAY_DINT[0][4] + 1;
    RETAINTEST_AUTO_STRUCTUREARRAYARRAY.ARRAYARRAY_DINT[0][5] := RETAINTEST_AUTO_STRUCTUREARRAYARRAY.ARRAYARRAY_DINT[0][5] + 1;
    RETAINTEST_AUTO_STRUCTUREARRAYARRAY.ARRAYARRAY_DINT[0][6] := RETAINTEST_AUTO_STRUCTUREARRAYARRAY.ARRAYARRAY_DINT[0][6] + 1;
    RETAINTEST_AUTO_STRUCTUREARRAYARRAY.ARRAYARRAY_DINT[0][7] := RETAINTEST_AUTO_STRUCTUREARRAYARRAY.ARRAYARRAY_DINT[0][7] + 1;
    RETAINTEST_AUTO_STRUCTUREARRAYARRAY.ARRAYARRAY_DINT[0][8] := RETAINTEST_AUTO_STRUCTUREARRAYARRAY.ARRAYARRAY_DINT[0][6];
    RETAINTEST_AUTO_STRUCTUREARRAYARRAY.ARRAYARRAY_DINT[0][9] := RETAINTEST_AUTO_STRUCTUREARRAYARRAY.ARRAYARRAY_DINT[0][7];

    RETAINTEST_AUTO_STRUCTUREARRAYARRAY.ARRAYARRAY_DINT[1][0] := RETAINTEST_AUTO_STRUCTUREARRAYARRAY.ARRAYARRAY_DINT[1][0] + 1;
    RETAINTEST_AUTO_STRUCTUREARRAYARRAY.ARRAYARRAY_DINT[1][1] := RETAINTEST_AUTO_STRUCTUREARRAYARRAY.ARRAYARRAY_DINT[1][1] + 1;
    RETAINTEST_AUTO_STRUCTUREARRAYARRAY.ARRAYARRAY_DINT[1][2] := RETAINTEST_AUTO_STRUCTUREARRAYARRAY.ARRAYARRAY_DINT[1][2] + 1;
    RETAINTEST_AUTO_STRUCTUREARRAYARRAY.ARRAYARRAY_DINT[1][3] := RETAINTEST_AUTO_STRUCTUREARRAYARRAY.ARRAYARRAY_DINT[1][3] + 1;
    RETAINTEST_AUTO_STRUCTUREARRAYARRAY.ARRAYARRAY_DINT[1][4] := RETAINTEST_AUTO_STRUCTUREARRAYARRAY.ARRAYARRAY_DINT[1][4] + 1;
    RETAINTEST_AUTO_STRUCTUREARRAYARRAY.ARRAYARRAY_DINT[1][5] := RETAINTEST_AUTO_STRUCTUREARRAYARRAY.ARRAYARRAY_DINT[1][5] + 1;
    RETAINTEST_AUTO_STRUCTUREARRAYARRAY.ARRAYARRAY_DINT[1][6] := RETAINTEST_AUTO_STRUCTUREARRAYARRAY.ARRAYARRAY_DINT[1][6] + 1;
    RETAINTEST_AUTO_STRUCTUREARRAYARRAY.ARRAYARRAY_DINT[1][7] := RETAINTEST_AUTO_STRUCTUREARRAYARRAY.ARRAYARRAY_DINT[1][7] + 1;
    RETAINTEST_AUTO_STRUCTUREARRAYARRAY.ARRAYARRAY_DINT[1][8] := RETAINTEST_AUTO_STRUCTUREARRAYARRAY.ARRAYARRAY_DINT[1][6];
    RETAINTEST_AUTO_STRUCTUREARRAYARRAY.ARRAYARRAY_DINT[1][9] := RETAINTEST_AUTO_STRUCTUREARRAYARRAY.ARRAYARRAY_DINT[1][7];

    RETAINTEST_AUTO_STRUCTUREARRAYARRAY.ARRAYARRAY_DINT[2][0] := RETAINTEST_AUTO_STRUCTUREARRAYARRAY.ARRAYARRAY_DINT[2][0] + 1;
    RETAINTEST_AUTO_STRUCTUREARRAYARRAY.ARRAYARRAY_DINT[2][1] := RETAINTEST_AUTO_STRUCTUREARRAYARRAY.ARRAYARRAY_DINT[2][1] + 1;
    RETAINTEST_AUTO_STRUCTUREARRAYARRAY.ARRAYARRAY_DINT[2][2] := RETAINTEST_AUTO_STRUCTUREARRAYARRAY.ARRAYARRAY_DINT[2][2] + 1;
    RETAINTEST_AUTO_STRUCTUREARRAYARRAY.ARRAYARRAY_DINT[2][3] := RETAINTEST_AUTO_STRUCTUREARRAYARRAY.ARRAYARRAY_DINT[2][3] + 1;
    RETAINTEST_AUTO_STRUCTUREARRAYARRAY.ARRAYARRAY_DINT[2][4] := RETAINTEST_AUTO_STRUCTUREARRAYARRAY.ARRAYARRAY_DINT[2][4] + 1;
    RETAINTEST_AUTO_STRUCTUREARRAYARRAY.ARRAYARRAY_DINT[2][5] := RETAINTEST_AUTO_STRUCTUREARRAYARRAY.ARRAYARRAY_DINT[2][5] + 1;
    RETAINTEST_AUTO_STRUCTUREARRAYARRAY.ARRAYARRAY_DINT[2][6] := RETAINTEST_AUTO_STRUCTUREARRAYARRAY.ARRAYARRAY_DINT[2][6] + 1;
    RETAINTEST_AUTO_STRUCTUREARRAYARRAY.ARRAYARRAY_DINT[2][7] := RETAINTEST_AUTO_STRUCTUREARRAYARRAY.ARRAYARRAY_DINT[2][7] + 1;
    RETAINTEST_AUTO_STRUCTUREARRAYARRAY.ARRAYARRAY_DINT[2][8] := RETAINTEST_AUTO_STRUCTUREARRAYARRAY.ARRAYARRAY_DINT[2][8] + 1;
    RETAINTEST_AUTO_STRUCTUREARRAYARRAY.ARRAYARRAY_DINT[2][9] := RETAINTEST_AUTO_STRUCTUREARRAYARRAY.ARRAYARRAY_DINT[2][9] + 1;

    RETAINTEST_AUTO_STRUCTUREARRAYARRAY.ARRAYARRAY_DINT[3][0] := RETAINTEST_AUTO_STRUCTUREARRAYARRAY.ARRAYARRAY_DINT[3][0] + 1;
    RETAINTEST_AUTO_STRUCTUREARRAYARRAY.ARRAYARRAY_DINT[3][1] := RETAINTEST_AUTO_STRUCTUREARRAYARRAY.ARRAYARRAY_DINT[3][1] + 1;
    RETAINTEST_AUTO_STRUCTUREARRAYARRAY.ARRAYARRAY_DINT[3][2] := RETAINTEST_AUTO_STRUCTUREARRAYARRAY.ARRAYARRAY_DINT[3][2] + 1;
    RETAINTEST_AUTO_STRUCTUREARRAYARRAY.ARRAYARRAY_DINT[3][3] := RETAINTEST_AUTO_STRUCTUREARRAYARRAY.ARRAYARRAY_DINT[3][3] + 1;
    RETAINTEST_AUTO_STRUCTUREARRAYARRAY.ARRAYARRAY_DINT[3][4] := RETAINTEST_AUTO_STRUCTUREARRAYARRAY.ARRAYARRAY_DINT[3][4] + 1;
    RETAINTEST_AUTO_STRUCTUREARRAYARRAY.ARRAYARRAY_DINT[3][5] := RETAINTEST_AUTO_STRUCTUREARRAYARRAY.ARRAYARRAY_DINT[3][5] + 1;
    RETAINTEST_AUTO_STRUCTUREARRAYARRAY.ARRAYARRAY_DINT[3][6] := RETAINTEST_AUTO_STRUCTUREARRAYARRAY.ARRAYARRAY_DINT[3][6] + 1;
    RETAINTEST_AUTO_STRUCTUREARRAYARRAY.ARRAYARRAY_DINT[3][7] := RETAINTEST_AUTO_STRUCTUREARRAYARRAY.ARRAYARRAY_DINT[3][7] + 1;
    RETAINTEST_AUTO_STRUCTUREARRAYARRAY.ARRAYARRAY_DINT[3][8] := RETAINTEST_AUTO_STRUCTUREARRAYARRAY.ARRAYARRAY_DINT[3][8] + 1;
    RETAINTEST_AUTO_STRUCTUREARRAYARRAY.ARRAYARRAY_DINT[3][9] := RETAINTEST_AUTO_STRUCTUREARRAYARRAY.ARRAYARRAY_DINT[3][9] + 1;

    RETAINTEST_AUTO_STRUCTUREARRAYARRAY.ARRAYARRAY_DINT[4][0] := RETAINTEST_AUTO_STRUCTUREARRAYARRAY.ARRAYARRAY_DINT[4][0] + 1;
    RETAINTEST_AUTO_STRUCTUREARRAYARRAY.ARRAYARRAY_DINT[4][1] := RETAINTEST_AUTO_STRUCTUREARRAYARRAY.ARRAYARRAY_DINT[4][1] + 1;
    RETAINTEST_AUTO_STRUCTUREARRAYARRAY.ARRAYARRAY_DINT[4][2] := RETAINTEST_AUTO_STRUCTUREARRAYARRAY.ARRAYARRAY_DINT[4][2] + 1;
    RETAINTEST_AUTO_STRUCTUREARRAYARRAY.ARRAYARRAY_DINT[4][3] := RETAINTEST_AUTO_STRUCTUREARRAYARRAY.ARRAYARRAY_DINT[4][3] + 1;
    RETAINTEST_AUTO_STRUCTUREARRAYARRAY.ARRAYARRAY_DINT[4][4] := RETAINTEST_AUTO_STRUCTUREARRAYARRAY.ARRAYARRAY_DINT[4][4] + 1;
    RETAINTEST_AUTO_STRUCTUREARRAYARRAY.ARRAYARRAY_DINT[4][5] := RETAINTEST_AUTO_STRUCTUREARRAYARRAY.ARRAYARRAY_DINT[4][5] + 1;
    RETAINTEST_AUTO_STRUCTUREARRAYARRAY.ARRAYARRAY_DINT[4][6] := RETAINTEST_AUTO_STRUCTUREARRAYARRAY.ARRAYARRAY_DINT[4][6] + 1;
    RETAINTEST_AUTO_STRUCTUREARRAYARRAY.ARRAYARRAY_DINT[4][7] := RETAINTEST_AUTO_STRUCTUREARRAYARRAY.ARRAYARRAY_DINT[4][7] + 1;
    RETAINTEST_AUTO_STRUCTUREARRAYARRAY.ARRAYARRAY_DINT[4][8] := RETAINTEST_AUTO_STRUCTUREARRAYARRAY.ARRAYARRAY_DINT[4][8] + 1;
    RETAINTEST_AUTO_STRUCTUREARRAYARRAY.ARRAYARRAY_DINT[4][9] := RETAINTEST_AUTO_STRUCTUREARRAYARRAY.ARRAYARRAY_DINT[4][9] + 1;

    RETAINTEST_AUTO_STRUCTUREARRAYARRAY.ARRAYARRAY_DINT[5][0] := RETAINTEST_AUTO_STRUCTUREARRAYARRAY.ARRAYARRAY_DINT[5][0] + 1;
    RETAINTEST_AUTO_STRUCTUREARRAYARRAY.ARRAYARRAY_DINT[5][1] := RETAINTEST_AUTO_STRUCTUREARRAYARRAY.ARRAYARRAY_DINT[5][1] + 1;
    RETAINTEST_AUTO_STRUCTUREARRAYARRAY.ARRAYARRAY_DINT[5][2] := RETAINTEST_AUTO_STRUCTUREARRAYARRAY.ARRAYARRAY_DINT[5][2] + 1;
    RETAINTEST_AUTO_STRUCTUREARRAYARRAY.ARRAYARRAY_DINT[5][3] := RETAINTEST_AUTO_STRUCTUREARRAYARRAY.ARRAYARRAY_DINT[5][3] + 1;
    RETAINTEST_AUTO_STRUCTUREARRAYARRAY.ARRAYARRAY_DINT[5][4] := RETAINTEST_AUTO_STRUCTUREARRAYARRAY.ARRAYARRAY_DINT[5][4] + 1;
    RETAINTEST_AUTO_STRUCTUREARRAYARRAY.ARRAYARRAY_DINT[5][5] := RETAINTEST_AUTO_STRUCTUREARRAYARRAY.ARRAYARRAY_DINT[5][5] + 1;
    RETAINTEST_AUTO_STRUCTUREARRAYARRAY.ARRAYARRAY_DINT[5][6] := RETAINTEST_AUTO_STRUCTUREARRAYARRAY.ARRAYARRAY_DINT[5][6] + 1;
    RETAINTEST_AUTO_STRUCTUREARRAYARRAY.ARRAYARRAY_DINT[5][7] := RETAINTEST_AUTO_STRUCTUREARRAYARRAY.ARRAYARRAY_DINT[5][7] + 1;
    RETAINTEST_AUTO_STRUCTUREARRAYARRAY.ARRAYARRAY_DINT[5][8] := RETAINTEST_AUTO_STRUCTUREARRAYARRAY.ARRAYARRAY_DINT[5][8] + 1;
    RETAINTEST_AUTO_STRUCTUREARRAYARRAY.ARRAYARRAY_DINT[5][9] := RETAINTEST_AUTO_STRUCTUREARRAYARRAY.ARRAYARRAY_DINT[5][9] + 1;

    RETAINTEST_AUTO_STRUCTUREARRAYARRAY.ARRAYARRAY_DINT[6][0] := RETAINTEST_AUTO_STRUCTUREARRAYARRAY.ARRAYARRAY_DINT[6][0] + 1;
    RETAINTEST_AUTO_STRUCTUREARRAYARRAY.ARRAYARRAY_DINT[6][1] := RETAINTEST_AUTO_STRUCTUREARRAYARRAY.ARRAYARRAY_DINT[6][1] + 1;
    RETAINTEST_AUTO_STRUCTUREARRAYARRAY.ARRAYARRAY_DINT[6][2] := RETAINTEST_AUTO_STRUCTUREARRAYARRAY.ARRAYARRAY_DINT[6][2] + 1;
    RETAINTEST_AUTO_STRUCTUREARRAYARRAY.ARRAYARRAY_DINT[6][3] := RETAINTEST_AUTO_STRUCTUREARRAYARRAY.ARRAYARRAY_DINT[6][3] + 1;
    RETAINTEST_AUTO_STRUCTUREARRAYARRAY.ARRAYARRAY_DINT[6][4] := RETAINTEST_AUTO_STRUCTUREARRAYARRAY.ARRAYARRAY_DINT[6][4] + 1;
    RETAINTEST_AUTO_STRUCTUREARRAYARRAY.ARRAYARRAY_DINT[6][5] := RETAINTEST_AUTO_STRUCTUREARRAYARRAY.ARRAYARRAY_DINT[6][5] + 1;
    RETAINTEST_AUTO_STRUCTUREARRAYARRAY.ARRAYARRAY_DINT[6][6] := RETAINTEST_AUTO_STRUCTUREARRAYARRAY.ARRAYARRAY_DINT[6][6] + 1;
    RETAINTEST_AUTO_STRUCTUREARRAYARRAY.ARRAYARRAY_DINT[6][7] := RETAINTEST_AUTO_STRUCTUREARRAYARRAY.ARRAYARRAY_DINT[6][7] + 1;
    RETAINTEST_AUTO_STRUCTUREARRAYARRAY.ARRAYARRAY_DINT[6][8] := RETAINTEST_AUTO_STRUCTUREARRAYARRAY.ARRAYARRAY_DINT[6][8] + 1;
    RETAINTEST_AUTO_STRUCTUREARRAYARRAY.ARRAYARRAY_DINT[6][9] := RETAINTEST_AUTO_STRUCTUREARRAYARRAY.ARRAYARRAY_DINT[6][9] + 1;

    RETAINTEST_AUTO_STRUCTUREARRAYARRAY.ARRAYARRAY_DINT[7][0] := RETAINTEST_AUTO_STRUCTUREARRAYARRAY.ARRAYARRAY_DINT[6][0];
    RETAINTEST_AUTO_STRUCTUREARRAYARRAY.ARRAYARRAY_DINT[7][1] := RETAINTEST_AUTO_STRUCTUREARRAYARRAY.ARRAYARRAY_DINT[6][1];
    RETAINTEST_AUTO_STRUCTUREARRAYARRAY.ARRAYARRAY_DINT[7][2] := RETAINTEST_AUTO_STRUCTUREARRAYARRAY.ARRAYARRAY_DINT[6][2];
    RETAINTEST_AUTO_STRUCTUREARRAYARRAY.ARRAYARRAY_DINT[7][3] := RETAINTEST_AUTO_STRUCTUREARRAYARRAY.ARRAYARRAY_DINT[6][3];
    RETAINTEST_AUTO_STRUCTUREARRAYARRAY.ARRAYARRAY_DINT[7][4] := RETAINTEST_AUTO_STRUCTUREARRAYARRAY.ARRAYARRAY_DINT[6][4];
    RETAINTEST_AUTO_STRUCTUREARRAYARRAY.ARRAYARRAY_DINT[7][5] := RETAINTEST_AUTO_STRUCTUREARRAYARRAY.ARRAYARRAY_DINT[6][5];
    RETAINTEST_AUTO_STRUCTUREARRAYARRAY.ARRAYARRAY_DINT[7][6] := RETAINTEST_AUTO_STRUCTUREARRAYARRAY.ARRAYARRAY_DINT[6][6];
    RETAINTEST_AUTO_STRUCTUREARRAYARRAY.ARRAYARRAY_DINT[7][7] := RETAINTEST_AUTO_STRUCTUREARRAYARRAY.ARRAYARRAY_DINT[6][7];
    RETAINTEST_AUTO_STRUCTUREARRAYARRAY.ARRAYARRAY_DINT[7][8] := RETAINTEST_AUTO_STRUCTUREARRAYARRAY.ARRAYARRAY_DINT[6][8];
    RETAINTEST_AUTO_STRUCTUREARRAYARRAY.ARRAYARRAY_DINT[7][9] := RETAINTEST_AUTO_STRUCTUREARRAYARRAY.ARRAYARRAY_DINT[6][9];

    RETAINTEST_AUTO_STRUCTUREARRAYARRAY.ARRAYARRAY_DWORD[0][0] := RETAINTEST_AUTO_STRUCTUREARRAYARRAY.ARRAYARRAY_DWORD[0][0] + 1;
    RETAINTEST_AUTO_STRUCTUREARRAYARRAY.ARRAYARRAY_DWORD[0][1] := RETAINTEST_AUTO_STRUCTUREARRAYARRAY.ARRAYARRAY_DWORD[0][1] + 1;
    RETAINTEST_AUTO_STRUCTUREARRAYARRAY.ARRAYARRAY_DWORD[0][2] := RETAINTEST_AUTO_STRUCTUREARRAYARRAY.ARRAYARRAY_DWORD[0][2] + 1;
    RETAINTEST_AUTO_STRUCTUREARRAYARRAY.ARRAYARRAY_DWORD[0][3] := RETAINTEST_AUTO_STRUCTUREARRAYARRAY.ARRAYARRAY_DWORD[0][3] + 1;
    RETAINTEST_AUTO_STRUCTUREARRAYARRAY.ARRAYARRAY_DWORD[0][4] := RETAINTEST_AUTO_STRUCTUREARRAYARRAY.ARRAYARRAY_DWORD[0][4] + 1;
    RETAINTEST_AUTO_STRUCTUREARRAYARRAY.ARRAYARRAY_DWORD[0][5] := RETAINTEST_AUTO_STRUCTUREARRAYARRAY.ARRAYARRAY_DWORD[0][5] + 1;
    RETAINTEST_AUTO_STRUCTUREARRAYARRAY.ARRAYARRAY_DWORD[0][6] := RETAINTEST_AUTO_STRUCTUREARRAYARRAY.ARRAYARRAY_DWORD[0][6] + 1;
    RETAINTEST_AUTO_STRUCTUREARRAYARRAY.ARRAYARRAY_DWORD[0][7] := RETAINTEST_AUTO_STRUCTUREARRAYARRAY.ARRAYARRAY_DWORD[0][7] + 1;
    RETAINTEST_AUTO_STRUCTUREARRAYARRAY.ARRAYARRAY_DWORD[0][8] := RETAINTEST_AUTO_STRUCTUREARRAYARRAY.ARRAYARRAY_DWORD[0][6];
    RETAINTEST_AUTO_STRUCTUREARRAYARRAY.ARRAYARRAY_DWORD[0][9] := RETAINTEST_AUTO_STRUCTUREARRAYARRAY.ARRAYARRAY_DWORD[0][7];

    RETAINTEST_AUTO_STRUCTUREARRAYARRAY.ARRAYARRAY_DWORD[1][0] := RETAINTEST_AUTO_STRUCTUREARRAYARRAY.ARRAYARRAY_DWORD[1][0] + 1;
    RETAINTEST_AUTO_STRUCTUREARRAYARRAY.ARRAYARRAY_DWORD[1][1] := RETAINTEST_AUTO_STRUCTUREARRAYARRAY.ARRAYARRAY_DWORD[1][1] + 1;
    RETAINTEST_AUTO_STRUCTUREARRAYARRAY.ARRAYARRAY_DWORD[1][2] := RETAINTEST_AUTO_STRUCTUREARRAYARRAY.ARRAYARRAY_DWORD[1][2] + 1;
    RETAINTEST_AUTO_STRUCTUREARRAYARRAY.ARRAYARRAY_DWORD[1][3] := RETAINTEST_AUTO_STRUCTUREARRAYARRAY.ARRAYARRAY_DWORD[1][3] + 1;
    RETAINTEST_AUTO_STRUCTUREARRAYARRAY.ARRAYARRAY_DWORD[1][4] := RETAINTEST_AUTO_STRUCTUREARRAYARRAY.ARRAYARRAY_DWORD[1][4] + 1;
    RETAINTEST_AUTO_STRUCTUREARRAYARRAY.ARRAYARRAY_DWORD[1][5] := RETAINTEST_AUTO_STRUCTUREARRAYARRAY.ARRAYARRAY_DWORD[1][5] + 1;
    RETAINTEST_AUTO_STRUCTUREARRAYARRAY.ARRAYARRAY_DWORD[1][6] := RETAINTEST_AUTO_STRUCTUREARRAYARRAY.ARRAYARRAY_DWORD[1][6] + 1;
    RETAINTEST_AUTO_STRUCTUREARRAYARRAY.ARRAYARRAY_DWORD[1][7] := RETAINTEST_AUTO_STRUCTUREARRAYARRAY.ARRAYARRAY_DWORD[1][7] + 1;
    RETAINTEST_AUTO_STRUCTUREARRAYARRAY.ARRAYARRAY_DWORD[1][8] := RETAINTEST_AUTO_STRUCTUREARRAYARRAY.ARRAYARRAY_DWORD[1][6];
    RETAINTEST_AUTO_STRUCTUREARRAYARRAY.ARRAYARRAY_DWORD[1][9] := RETAINTEST_AUTO_STRUCTUREARRAYARRAY.ARRAYARRAY_DWORD[1][7];

    RETAINTEST_AUTO_STRUCTUREARRAYARRAY.ARRAYARRAY_DWORD[2][0] := RETAINTEST_AUTO_STRUCTUREARRAYARRAY.ARRAYARRAY_DWORD[2][0] + 1;
    RETAINTEST_AUTO_STRUCTUREARRAYARRAY.ARRAYARRAY_DWORD[2][1] := RETAINTEST_AUTO_STRUCTUREARRAYARRAY.ARRAYARRAY_DWORD[2][1] + 1;
    RETAINTEST_AUTO_STRUCTUREARRAYARRAY.ARRAYARRAY_DWORD[2][2] := RETAINTEST_AUTO_STRUCTUREARRAYARRAY.ARRAYARRAY_DWORD[2][2] + 1;
    RETAINTEST_AUTO_STRUCTUREARRAYARRAY.ARRAYARRAY_DWORD[2][3] := RETAINTEST_AUTO_STRUCTUREARRAYARRAY.ARRAYARRAY_DWORD[2][3] + 1;
    RETAINTEST_AUTO_STRUCTUREARRAYARRAY.ARRAYARRAY_DWORD[2][4] := RETAINTEST_AUTO_STRUCTUREARRAYARRAY.ARRAYARRAY_DWORD[2][4] + 1;
    RETAINTEST_AUTO_STRUCTUREARRAYARRAY.ARRAYARRAY_DWORD[2][5] := RETAINTEST_AUTO_STRUCTUREARRAYARRAY.ARRAYARRAY_DWORD[2][5] + 1;
    RETAINTEST_AUTO_STRUCTUREARRAYARRAY.ARRAYARRAY_DWORD[2][6] := RETAINTEST_AUTO_STRUCTUREARRAYARRAY.ARRAYARRAY_DWORD[2][6] + 1;
    RETAINTEST_AUTO_STRUCTUREARRAYARRAY.ARRAYARRAY_DWORD[2][7] := RETAINTEST_AUTO_STRUCTUREARRAYARRAY.ARRAYARRAY_DWORD[2][7] + 1;
    RETAINTEST_AUTO_STRUCTUREARRAYARRAY.ARRAYARRAY_DWORD[2][8] := RETAINTEST_AUTO_STRUCTUREARRAYARRAY.ARRAYARRAY_DWORD[2][8] + 1;
    RETAINTEST_AUTO_STRUCTUREARRAYARRAY.ARRAYARRAY_DWORD[2][9] := RETAINTEST_AUTO_STRUCTUREARRAYARRAY.ARRAYARRAY_DWORD[2][9] + 1;

    RETAINTEST_AUTO_STRUCTUREARRAYARRAY.ARRAYARRAY_DWORD[3][0] := RETAINTEST_AUTO_STRUCTUREARRAYARRAY.ARRAYARRAY_DWORD[3][0] + 1;
    RETAINTEST_AUTO_STRUCTUREARRAYARRAY.ARRAYARRAY_DWORD[3][1] := RETAINTEST_AUTO_STRUCTUREARRAYARRAY.ARRAYARRAY_DWORD[3][1] + 1;
    RETAINTEST_AUTO_STRUCTUREARRAYARRAY.ARRAYARRAY_DWORD[3][2] := RETAINTEST_AUTO_STRUCTUREARRAYARRAY.ARRAYARRAY_DWORD[3][2] + 1;
    RETAINTEST_AUTO_STRUCTUREARRAYARRAY.ARRAYARRAY_DWORD[3][3] := RETAINTEST_AUTO_STRUCTUREARRAYARRAY.ARRAYARRAY_DWORD[3][3] + 1;
    RETAINTEST_AUTO_STRUCTUREARRAYARRAY.ARRAYARRAY_DWORD[3][4] := RETAINTEST_AUTO_STRUCTUREARRAYARRAY.ARRAYARRAY_DWORD[3][4] + 1;
    RETAINTEST_AUTO_STRUCTUREARRAYARRAY.ARRAYARRAY_DWORD[3][5] := RETAINTEST_AUTO_STRUCTUREARRAYARRAY.ARRAYARRAY_DWORD[3][5] + 1;
    RETAINTEST_AUTO_STRUCTUREARRAYARRAY.ARRAYARRAY_DWORD[3][6] := RETAINTEST_AUTO_STRUCTUREARRAYARRAY.ARRAYARRAY_DWORD[3][6] + 1;
    RETAINTEST_AUTO_STRUCTUREARRAYARRAY.ARRAYARRAY_DWORD[3][7] := RETAINTEST_AUTO_STRUCTUREARRAYARRAY.ARRAYARRAY_DWORD[3][7] + 1;
    RETAINTEST_AUTO_STRUCTUREARRAYARRAY.ARRAYARRAY_DWORD[3][8] := RETAINTEST_AUTO_STRUCTUREARRAYARRAY.ARRAYARRAY_DWORD[3][8] + 1;
    RETAINTEST_AUTO_STRUCTUREARRAYARRAY.ARRAYARRAY_DWORD[3][9] := RETAINTEST_AUTO_STRUCTUREARRAYARRAY.ARRAYARRAY_DWORD[3][9] + 1;

    RETAINTEST_AUTO_STRUCTUREARRAYARRAY.ARRAYARRAY_DWORD[4][0] := RETAINTEST_AUTO_STRUCTUREARRAYARRAY.ARRAYARRAY_DWORD[4][0] + 1;
    RETAINTEST_AUTO_STRUCTUREARRAYARRAY.ARRAYARRAY_DWORD[4][1] := RETAINTEST_AUTO_STRUCTUREARRAYARRAY.ARRAYARRAY_DWORD[4][1] + 1;
    RETAINTEST_AUTO_STRUCTUREARRAYARRAY.ARRAYARRAY_DWORD[4][2] := RETAINTEST_AUTO_STRUCTUREARRAYARRAY.ARRAYARRAY_DWORD[4][2] + 1;
    RETAINTEST_AUTO_STRUCTUREARRAYARRAY.ARRAYARRAY_DWORD[4][3] := RETAINTEST_AUTO_STRUCTUREARRAYARRAY.ARRAYARRAY_DWORD[4][3] + 1;
    RETAINTEST_AUTO_STRUCTUREARRAYARRAY.ARRAYARRAY_DWORD[4][4] := RETAINTEST_AUTO_STRUCTUREARRAYARRAY.ARRAYARRAY_DWORD[4][4] + 1;
    RETAINTEST_AUTO_STRUCTUREARRAYARRAY.ARRAYARRAY_DWORD[4][5] := RETAINTEST_AUTO_STRUCTUREARRAYARRAY.ARRAYARRAY_DWORD[4][5] + 1;
    RETAINTEST_AUTO_STRUCTUREARRAYARRAY.ARRAYARRAY_DWORD[4][6] := RETAINTEST_AUTO_STRUCTUREARRAYARRAY.ARRAYARRAY_DWORD[4][6] + 1;
    RETAINTEST_AUTO_STRUCTUREARRAYARRAY.ARRAYARRAY_DWORD[4][7] := RETAINTEST_AUTO_STRUCTUREARRAYARRAY.ARRAYARRAY_DWORD[4][7] + 1;
    RETAINTEST_AUTO_STRUCTUREARRAYARRAY.ARRAYARRAY_DWORD[4][8] := RETAINTEST_AUTO_STRUCTUREARRAYARRAY.ARRAYARRAY_DWORD[4][8] + 1;
    RETAINTEST_AUTO_STRUCTUREARRAYARRAY.ARRAYARRAY_DWORD[4][9] := RETAINTEST_AUTO_STRUCTUREARRAYARRAY.ARRAYARRAY_DWORD[4][9] + 1;

    RETAINTEST_AUTO_STRUCTUREARRAYARRAY.ARRAYARRAY_DWORD[5][0] := RETAINTEST_AUTO_STRUCTUREARRAYARRAY.ARRAYARRAY_DWORD[5][0] + 1;
    RETAINTEST_AUTO_STRUCTUREARRAYARRAY.ARRAYARRAY_DWORD[5][1] := RETAINTEST_AUTO_STRUCTUREARRAYARRAY.ARRAYARRAY_DWORD[5][1] + 1;
    RETAINTEST_AUTO_STRUCTUREARRAYARRAY.ARRAYARRAY_DWORD[5][2] := RETAINTEST_AUTO_STRUCTUREARRAYARRAY.ARRAYARRAY_DWORD[5][2] + 1;
    RETAINTEST_AUTO_STRUCTUREARRAYARRAY.ARRAYARRAY_DWORD[5][3] := RETAINTEST_AUTO_STRUCTUREARRAYARRAY.ARRAYARRAY_DWORD[5][3] + 1;
    RETAINTEST_AUTO_STRUCTUREARRAYARRAY.ARRAYARRAY_DWORD[5][4] := RETAINTEST_AUTO_STRUCTUREARRAYARRAY.ARRAYARRAY_DWORD[5][4] + 1;
    RETAINTEST_AUTO_STRUCTUREARRAYARRAY.ARRAYARRAY_DWORD[5][5] := RETAINTEST_AUTO_STRUCTUREARRAYARRAY.ARRAYARRAY_DWORD[5][5] + 1;
    RETAINTEST_AUTO_STRUCTUREARRAYARRAY.ARRAYARRAY_DWORD[5][6] := RETAINTEST_AUTO_STRUCTUREARRAYARRAY.ARRAYARRAY_DWORD[5][6] + 1;
    RETAINTEST_AUTO_STRUCTUREARRAYARRAY.ARRAYARRAY_DWORD[5][7] := RETAINTEST_AUTO_STRUCTUREARRAYARRAY.ARRAYARRAY_DWORD[5][7] + 1;
    RETAINTEST_AUTO_STRUCTUREARRAYARRAY.ARRAYARRAY_DWORD[5][8] := RETAINTEST_AUTO_STRUCTUREARRAYARRAY.ARRAYARRAY_DWORD[5][8] + 1;
    RETAINTEST_AUTO_STRUCTUREARRAYARRAY.ARRAYARRAY_DWORD[5][9] := RETAINTEST_AUTO_STRUCTUREARRAYARRAY.ARRAYARRAY_DWORD[5][9] + 1;

    RETAINTEST_AUTO_STRUCTUREARRAYARRAY.ARRAYARRAY_DWORD[6][0] := RETAINTEST_AUTO_STRUCTUREARRAYARRAY.ARRAYARRAY_DWORD[6][0] + 1;
    RETAINTEST_AUTO_STRUCTUREARRAYARRAY.ARRAYARRAY_DWORD[6][1] := RETAINTEST_AUTO_STRUCTUREARRAYARRAY.ARRAYARRAY_DWORD[6][1] + 1;
    RETAINTEST_AUTO_STRUCTUREARRAYARRAY.ARRAYARRAY_DWORD[6][2] := RETAINTEST_AUTO_STRUCTUREARRAYARRAY.ARRAYARRAY_DWORD[6][2] + 1;
    RETAINTEST_AUTO_STRUCTUREARRAYARRAY.ARRAYARRAY_DWORD[6][3] := RETAINTEST_AUTO_STRUCTUREARRAYARRAY.ARRAYARRAY_DWORD[6][3] + 1;
    RETAINTEST_AUTO_STRUCTUREARRAYARRAY.ARRAYARRAY_DWORD[6][4] := RETAINTEST_AUTO_STRUCTUREARRAYARRAY.ARRAYARRAY_DWORD[6][4] + 1;
    RETAINTEST_AUTO_STRUCTUREARRAYARRAY.ARRAYARRAY_DWORD[6][5] := RETAINTEST_AUTO_STRUCTUREARRAYARRAY.ARRAYARRAY_DWORD[6][5] + 1;
    RETAINTEST_AUTO_STRUCTUREARRAYARRAY.ARRAYARRAY_DWORD[6][6] := RETAINTEST_AUTO_STRUCTUREARRAYARRAY.ARRAYARRAY_DWORD[6][6] + 1;
    RETAINTEST_AUTO_STRUCTUREARRAYARRAY.ARRAYARRAY_DWORD[6][7] := RETAINTEST_AUTO_STRUCTUREARRAYARRAY.ARRAYARRAY_DWORD[6][7] + 1;
    RETAINTEST_AUTO_STRUCTUREARRAYARRAY.ARRAYARRAY_DWORD[6][8] := RETAINTEST_AUTO_STRUCTUREARRAYARRAY.ARRAYARRAY_DWORD[6][8] + 1;
    RETAINTEST_AUTO_STRUCTUREARRAYARRAY.ARRAYARRAY_DWORD[6][9] := RETAINTEST_AUTO_STRUCTUREARRAYARRAY.ARRAYARRAY_DWORD[6][9] + 1;

    RETAINTEST_AUTO_STRUCTUREARRAYARRAY.ARRAYARRAY_DWORD[7][0] := RETAINTEST_AUTO_STRUCTUREARRAYARRAY.ARRAYARRAY_DWORD[6][0];
    RETAINTEST_AUTO_STRUCTUREARRAYARRAY.ARRAYARRAY_DWORD[7][1] := RETAINTEST_AUTO_STRUCTUREARRAYARRAY.ARRAYARRAY_DWORD[6][1];
    RETAINTEST_AUTO_STRUCTUREARRAYARRAY.ARRAYARRAY_DWORD[7][2] := RETAINTEST_AUTO_STRUCTUREARRAYARRAY.ARRAYARRAY_DWORD[6][2];
    RETAINTEST_AUTO_STRUCTUREARRAYARRAY.ARRAYARRAY_DWORD[7][3] := RETAINTEST_AUTO_STRUCTUREARRAYARRAY.ARRAYARRAY_DWORD[6][3];
    RETAINTEST_AUTO_STRUCTUREARRAYARRAY.ARRAYARRAY_DWORD[7][4] := RETAINTEST_AUTO_STRUCTUREARRAYARRAY.ARRAYARRAY_DWORD[6][4];
    RETAINTEST_AUTO_STRUCTUREARRAYARRAY.ARRAYARRAY_DWORD[7][5] := RETAINTEST_AUTO_STRUCTUREARRAYARRAY.ARRAYARRAY_DWORD[6][5];
    RETAINTEST_AUTO_STRUCTUREARRAYARRAY.ARRAYARRAY_DWORD[7][6] := RETAINTEST_AUTO_STRUCTUREARRAYARRAY.ARRAYARRAY_DWORD[6][6];
    RETAINTEST_AUTO_STRUCTUREARRAYARRAY.ARRAYARRAY_DWORD[7][7] := RETAINTEST_AUTO_STRUCTUREARRAYARRAY.ARRAYARRAY_DWORD[6][7];
    RETAINTEST_AUTO_STRUCTUREARRAYARRAY.ARRAYARRAY_DWORD[7][8] := RETAINTEST_AUTO_STRUCTUREARRAYARRAY.ARRAYARRAY_DWORD[6][8];
    RETAINTEST_AUTO_STRUCTUREARRAYARRAY.ARRAYARRAY_DWORD[7][9] := RETAINTEST_AUTO_STRUCTUREARRAYARRAY.ARRAYARRAY_DWORD[6][9];

    RETAINTEST_AUTO_STRUCTUREARRAYARRAY.ARRAYARRAY_INT[0][0] := RETAINTEST_AUTO_STRUCTUREARRAYARRAY.ARRAYARRAY_INT[0][0] + 1;
    RETAINTEST_AUTO_STRUCTUREARRAYARRAY.ARRAYARRAY_INT[0][1] := RETAINTEST_AUTO_STRUCTUREARRAYARRAY.ARRAYARRAY_INT[0][1] + 1;
    RETAINTEST_AUTO_STRUCTUREARRAYARRAY.ARRAYARRAY_INT[0][2] := RETAINTEST_AUTO_STRUCTUREARRAYARRAY.ARRAYARRAY_INT[0][2] + 1;
    RETAINTEST_AUTO_STRUCTUREARRAYARRAY.ARRAYARRAY_INT[0][3] := RETAINTEST_AUTO_STRUCTUREARRAYARRAY.ARRAYARRAY_INT[0][3] + 1;
    RETAINTEST_AUTO_STRUCTUREARRAYARRAY.ARRAYARRAY_INT[0][4] := RETAINTEST_AUTO_STRUCTUREARRAYARRAY.ARRAYARRAY_INT[0][4] + 1;
    RETAINTEST_AUTO_STRUCTUREARRAYARRAY.ARRAYARRAY_INT[0][5] := RETAINTEST_AUTO_STRUCTUREARRAYARRAY.ARRAYARRAY_INT[0][5] + 1;
    RETAINTEST_AUTO_STRUCTUREARRAYARRAY.ARRAYARRAY_INT[0][6] := RETAINTEST_AUTO_STRUCTUREARRAYARRAY.ARRAYARRAY_INT[0][6] + 1;
    RETAINTEST_AUTO_STRUCTUREARRAYARRAY.ARRAYARRAY_INT[0][7] := RETAINTEST_AUTO_STRUCTUREARRAYARRAY.ARRAYARRAY_INT[0][7] + 1;
    RETAINTEST_AUTO_STRUCTUREARRAYARRAY.ARRAYARRAY_INT[0][8] := RETAINTEST_AUTO_STRUCTUREARRAYARRAY.ARRAYARRAY_INT[0][6];
    RETAINTEST_AUTO_STRUCTUREARRAYARRAY.ARRAYARRAY_INT[0][9] := RETAINTEST_AUTO_STRUCTUREARRAYARRAY.ARRAYARRAY_INT[0][7];

    RETAINTEST_AUTO_STRUCTUREARRAYARRAY.ARRAYARRAY_INT[1][0] := RETAINTEST_AUTO_STRUCTUREARRAYARRAY.ARRAYARRAY_INT[1][0] + 1;
    RETAINTEST_AUTO_STRUCTUREARRAYARRAY.ARRAYARRAY_INT[1][1] := RETAINTEST_AUTO_STRUCTUREARRAYARRAY.ARRAYARRAY_INT[1][1] + 1;
    RETAINTEST_AUTO_STRUCTUREARRAYARRAY.ARRAYARRAY_INT[1][2] := RETAINTEST_AUTO_STRUCTUREARRAYARRAY.ARRAYARRAY_INT[1][2] + 1;
    RETAINTEST_AUTO_STRUCTUREARRAYARRAY.ARRAYARRAY_INT[1][3] := RETAINTEST_AUTO_STRUCTUREARRAYARRAY.ARRAYARRAY_INT[1][3] + 1;
    RETAINTEST_AUTO_STRUCTUREARRAYARRAY.ARRAYARRAY_INT[1][4] := RETAINTEST_AUTO_STRUCTUREARRAYARRAY.ARRAYARRAY_INT[1][4] + 1;
    RETAINTEST_AUTO_STRUCTUREARRAYARRAY.ARRAYARRAY_INT[1][5] := RETAINTEST_AUTO_STRUCTUREARRAYARRAY.ARRAYARRAY_INT[1][5] + 1;
    RETAINTEST_AUTO_STRUCTUREARRAYARRAY.ARRAYARRAY_INT[1][6] := RETAINTEST_AUTO_STRUCTUREARRAYARRAY.ARRAYARRAY_INT[1][6] + 1;
    RETAINTEST_AUTO_STRUCTUREARRAYARRAY.ARRAYARRAY_INT[1][7] := RETAINTEST_AUTO_STRUCTUREARRAYARRAY.ARRAYARRAY_INT[1][7] + 1;
    RETAINTEST_AUTO_STRUCTUREARRAYARRAY.ARRAYARRAY_INT[1][8] := RETAINTEST_AUTO_STRUCTUREARRAYARRAY.ARRAYARRAY_INT[1][6];
    RETAINTEST_AUTO_STRUCTUREARRAYARRAY.ARRAYARRAY_INT[1][9] := RETAINTEST_AUTO_STRUCTUREARRAYARRAY.ARRAYARRAY_INT[1][7];

    RETAINTEST_AUTO_STRUCTUREARRAYARRAY.ARRAYARRAY_INT[2][0] := RETAINTEST_AUTO_STRUCTUREARRAYARRAY.ARRAYARRAY_INT[2][0] + 1;
    RETAINTEST_AUTO_STRUCTUREARRAYARRAY.ARRAYARRAY_INT[2][1] := RETAINTEST_AUTO_STRUCTUREARRAYARRAY.ARRAYARRAY_INT[2][1] + 1;
    RETAINTEST_AUTO_STRUCTUREARRAYARRAY.ARRAYARRAY_INT[2][2] := RETAINTEST_AUTO_STRUCTUREARRAYARRAY.ARRAYARRAY_INT[2][2] + 1;
    RETAINTEST_AUTO_STRUCTUREARRAYARRAY.ARRAYARRAY_INT[2][3] := RETAINTEST_AUTO_STRUCTUREARRAYARRAY.ARRAYARRAY_INT[2][3] + 1;
    RETAINTEST_AUTO_STRUCTUREARRAYARRAY.ARRAYARRAY_INT[2][4] := RETAINTEST_AUTO_STRUCTUREARRAYARRAY.ARRAYARRAY_INT[2][4] + 1;
    RETAINTEST_AUTO_STRUCTUREARRAYARRAY.ARRAYARRAY_INT[2][5] := RETAINTEST_AUTO_STRUCTUREARRAYARRAY.ARRAYARRAY_INT[2][5] + 1;
    RETAINTEST_AUTO_STRUCTUREARRAYARRAY.ARRAYARRAY_INT[2][6] := RETAINTEST_AUTO_STRUCTUREARRAYARRAY.ARRAYARRAY_INT[2][6] + 1;
    RETAINTEST_AUTO_STRUCTUREARRAYARRAY.ARRAYARRAY_INT[2][7] := RETAINTEST_AUTO_STRUCTUREARRAYARRAY.ARRAYARRAY_INT[2][7] + 1;
    RETAINTEST_AUTO_STRUCTUREARRAYARRAY.ARRAYARRAY_INT[2][8] := RETAINTEST_AUTO_STRUCTUREARRAYARRAY.ARRAYARRAY_INT[2][8] + 1;
    RETAINTEST_AUTO_STRUCTUREARRAYARRAY.ARRAYARRAY_INT[2][9] := RETAINTEST_AUTO_STRUCTUREARRAYARRAY.ARRAYARRAY_INT[2][9] + 1;

    RETAINTEST_AUTO_STRUCTUREARRAYARRAY.ARRAYARRAY_INT[3][0] := RETAINTEST_AUTO_STRUCTUREARRAYARRAY.ARRAYARRAY_INT[3][0] + 1;
    RETAINTEST_AUTO_STRUCTUREARRAYARRAY.ARRAYARRAY_INT[3][1] := RETAINTEST_AUTO_STRUCTUREARRAYARRAY.ARRAYARRAY_INT[3][1] + 1;
    RETAINTEST_AUTO_STRUCTUREARRAYARRAY.ARRAYARRAY_INT[3][2] := RETAINTEST_AUTO_STRUCTUREARRAYARRAY.ARRAYARRAY_INT[3][2] + 1;
    RETAINTEST_AUTO_STRUCTUREARRAYARRAY.ARRAYARRAY_INT[3][3] := RETAINTEST_AUTO_STRUCTUREARRAYARRAY.ARRAYARRAY_INT[3][3] + 1;
    RETAINTEST_AUTO_STRUCTUREARRAYARRAY.ARRAYARRAY_INT[3][4] := RETAINTEST_AUTO_STRUCTUREARRAYARRAY.ARRAYARRAY_INT[3][4] + 1;
    RETAINTEST_AUTO_STRUCTUREARRAYARRAY.ARRAYARRAY_INT[3][5] := RETAINTEST_AUTO_STRUCTUREARRAYARRAY.ARRAYARRAY_INT[3][5] + 1;
    RETAINTEST_AUTO_STRUCTUREARRAYARRAY.ARRAYARRAY_INT[3][6] := RETAINTEST_AUTO_STRUCTUREARRAYARRAY.ARRAYARRAY_INT[3][6] + 1;
    RETAINTEST_AUTO_STRUCTUREARRAYARRAY.ARRAYARRAY_INT[3][7] := RETAINTEST_AUTO_STRUCTUREARRAYARRAY.ARRAYARRAY_INT[3][7] + 1;
    RETAINTEST_AUTO_STRUCTUREARRAYARRAY.ARRAYARRAY_INT[3][8] := RETAINTEST_AUTO_STRUCTUREARRAYARRAY.ARRAYARRAY_INT[3][8] + 1;
    RETAINTEST_AUTO_STRUCTUREARRAYARRAY.ARRAYARRAY_INT[3][9] := RETAINTEST_AUTO_STRUCTUREARRAYARRAY.ARRAYARRAY_INT[3][9] + 1;

    RETAINTEST_AUTO_STRUCTUREARRAYARRAY.ARRAYARRAY_INT[4][0] := RETAINTEST_AUTO_STRUCTUREARRAYARRAY.ARRAYARRAY_INT[4][0] + 1;
    RETAINTEST_AUTO_STRUCTUREARRAYARRAY.ARRAYARRAY_INT[4][1] := RETAINTEST_AUTO_STRUCTUREARRAYARRAY.ARRAYARRAY_INT[4][1] + 1;
    RETAINTEST_AUTO_STRUCTUREARRAYARRAY.ARRAYARRAY_INT[4][2] := RETAINTEST_AUTO_STRUCTUREARRAYARRAY.ARRAYARRAY_INT[4][2] + 1;
    RETAINTEST_AUTO_STRUCTUREARRAYARRAY.ARRAYARRAY_INT[4][3] := RETAINTEST_AUTO_STRUCTUREARRAYARRAY.ARRAYARRAY_INT[4][3] + 1;
    RETAINTEST_AUTO_STRUCTUREARRAYARRAY.ARRAYARRAY_INT[4][4] := RETAINTEST_AUTO_STRUCTUREARRAYARRAY.ARRAYARRAY_INT[4][4] + 1;
    RETAINTEST_AUTO_STRUCTUREARRAYARRAY.ARRAYARRAY_INT[4][5] := RETAINTEST_AUTO_STRUCTUREARRAYARRAY.ARRAYARRAY_INT[4][5] + 1;
    RETAINTEST_AUTO_STRUCTUREARRAYARRAY.ARRAYARRAY_INT[4][6] := RETAINTEST_AUTO_STRUCTUREARRAYARRAY.ARRAYARRAY_INT[4][6] + 1;
    RETAINTEST_AUTO_STRUCTUREARRAYARRAY.ARRAYARRAY_INT[4][7] := RETAINTEST_AUTO_STRUCTUREARRAYARRAY.ARRAYARRAY_INT[4][7] + 1;
    RETAINTEST_AUTO_STRUCTUREARRAYARRAY.ARRAYARRAY_INT[4][8] := RETAINTEST_AUTO_STRUCTUREARRAYARRAY.ARRAYARRAY_INT[4][8] + 1;
    RETAINTEST_AUTO_STRUCTUREARRAYARRAY.ARRAYARRAY_INT[4][9] := RETAINTEST_AUTO_STRUCTUREARRAYARRAY.ARRAYARRAY_INT[4][9] + 1;

    RETAINTEST_AUTO_STRUCTUREARRAYARRAY.ARRAYARRAY_INT[5][0] := RETAINTEST_AUTO_STRUCTUREARRAYARRAY.ARRAYARRAY_INT[5][0] + 1;
    RETAINTEST_AUTO_STRUCTUREARRAYARRAY.ARRAYARRAY_INT[5][1] := RETAINTEST_AUTO_STRUCTUREARRAYARRAY.ARRAYARRAY_INT[5][1] + 1;
    RETAINTEST_AUTO_STRUCTUREARRAYARRAY.ARRAYARRAY_INT[5][2] := RETAINTEST_AUTO_STRUCTUREARRAYARRAY.ARRAYARRAY_INT[5][2] + 1;
    RETAINTEST_AUTO_STRUCTUREARRAYARRAY.ARRAYARRAY_INT[5][3] := RETAINTEST_AUTO_STRUCTUREARRAYARRAY.ARRAYARRAY_INT[5][3] + 1;
    RETAINTEST_AUTO_STRUCTUREARRAYARRAY.ARRAYARRAY_INT[5][4] := RETAINTEST_AUTO_STRUCTUREARRAYARRAY.ARRAYARRAY_INT[5][4] + 1;
    RETAINTEST_AUTO_STRUCTUREARRAYARRAY.ARRAYARRAY_INT[5][5] := RETAINTEST_AUTO_STRUCTUREARRAYARRAY.ARRAYARRAY_INT[5][5] + 1;
    RETAINTEST_AUTO_STRUCTUREARRAYARRAY.ARRAYARRAY_INT[5][6] := RETAINTEST_AUTO_STRUCTUREARRAYARRAY.ARRAYARRAY_INT[5][6] + 1;
    RETAINTEST_AUTO_STRUCTUREARRAYARRAY.ARRAYARRAY_INT[5][7] := RETAINTEST_AUTO_STRUCTUREARRAYARRAY.ARRAYARRAY_INT[5][7] + 1;
    RETAINTEST_AUTO_STRUCTUREARRAYARRAY.ARRAYARRAY_INT[5][8] := RETAINTEST_AUTO_STRUCTUREARRAYARRAY.ARRAYARRAY_INT[5][8] + 1;
    RETAINTEST_AUTO_STRUCTUREARRAYARRAY.ARRAYARRAY_INT[5][9] := RETAINTEST_AUTO_STRUCTUREARRAYARRAY.ARRAYARRAY_INT[5][9] + 1;

    RETAINTEST_AUTO_STRUCTUREARRAYARRAY.ARRAYARRAY_INT[6][0] := RETAINTEST_AUTO_STRUCTUREARRAYARRAY.ARRAYARRAY_INT[6][0] + 1;
    RETAINTEST_AUTO_STRUCTUREARRAYARRAY.ARRAYARRAY_INT[6][1] := RETAINTEST_AUTO_STRUCTUREARRAYARRAY.ARRAYARRAY_INT[6][1] + 1;
    RETAINTEST_AUTO_STRUCTUREARRAYARRAY.ARRAYARRAY_INT[6][2] := RETAINTEST_AUTO_STRUCTUREARRAYARRAY.ARRAYARRAY_INT[6][2] + 1;
    RETAINTEST_AUTO_STRUCTUREARRAYARRAY.ARRAYARRAY_INT[6][3] := RETAINTEST_AUTO_STRUCTUREARRAYARRAY.ARRAYARRAY_INT[6][3] + 1;
    RETAINTEST_AUTO_STRUCTUREARRAYARRAY.ARRAYARRAY_INT[6][4] := RETAINTEST_AUTO_STRUCTUREARRAYARRAY.ARRAYARRAY_INT[6][4] + 1;
    RETAINTEST_AUTO_STRUCTUREARRAYARRAY.ARRAYARRAY_INT[6][5] := RETAINTEST_AUTO_STRUCTUREARRAYARRAY.ARRAYARRAY_INT[6][5] + 1;
    RETAINTEST_AUTO_STRUCTUREARRAYARRAY.ARRAYARRAY_INT[6][6] := RETAINTEST_AUTO_STRUCTUREARRAYARRAY.ARRAYARRAY_INT[6][6] + 1;
    RETAINTEST_AUTO_STRUCTUREARRAYARRAY.ARRAYARRAY_INT[6][7] := RETAINTEST_AUTO_STRUCTUREARRAYARRAY.ARRAYARRAY_INT[6][7] + 1;
    RETAINTEST_AUTO_STRUCTUREARRAYARRAY.ARRAYARRAY_INT[6][8] := RETAINTEST_AUTO_STRUCTUREARRAYARRAY.ARRAYARRAY_INT[6][8] + 1;
    RETAINTEST_AUTO_STRUCTUREARRAYARRAY.ARRAYARRAY_INT[6][9] := RETAINTEST_AUTO_STRUCTUREARRAYARRAY.ARRAYARRAY_INT[6][9] + 1;

    RETAINTEST_AUTO_STRUCTUREARRAYARRAY.ARRAYARRAY_INT[7][0] := RETAINTEST_AUTO_STRUCTUREARRAYARRAY.ARRAYARRAY_INT[6][0];
    RETAINTEST_AUTO_STRUCTUREARRAYARRAY.ARRAYARRAY_INT[7][1] := RETAINTEST_AUTO_STRUCTUREARRAYARRAY.ARRAYARRAY_INT[6][1];
    RETAINTEST_AUTO_STRUCTUREARRAYARRAY.ARRAYARRAY_INT[7][2] := RETAINTEST_AUTO_STRUCTUREARRAYARRAY.ARRAYARRAY_INT[6][2];
    RETAINTEST_AUTO_STRUCTUREARRAYARRAY.ARRAYARRAY_INT[7][3] := RETAINTEST_AUTO_STRUCTUREARRAYARRAY.ARRAYARRAY_INT[6][3];
    RETAINTEST_AUTO_STRUCTUREARRAYARRAY.ARRAYARRAY_INT[7][4] := RETAINTEST_AUTO_STRUCTUREARRAYARRAY.ARRAYARRAY_INT[6][4];
    RETAINTEST_AUTO_STRUCTUREARRAYARRAY.ARRAYARRAY_INT[7][5] := RETAINTEST_AUTO_STRUCTUREARRAYARRAY.ARRAYARRAY_INT[6][5];
    RETAINTEST_AUTO_STRUCTUREARRAYARRAY.ARRAYARRAY_INT[7][6] := RETAINTEST_AUTO_STRUCTUREARRAYARRAY.ARRAYARRAY_INT[6][6];
    RETAINTEST_AUTO_STRUCTUREARRAYARRAY.ARRAYARRAY_INT[7][7] := RETAINTEST_AUTO_STRUCTUREARRAYARRAY.ARRAYARRAY_INT[6][7];
    RETAINTEST_AUTO_STRUCTUREARRAYARRAY.ARRAYARRAY_INT[7][8] := RETAINTEST_AUTO_STRUCTUREARRAYARRAY.ARRAYARRAY_INT[6][8];
    RETAINTEST_AUTO_STRUCTUREARRAYARRAY.ARRAYARRAY_INT[7][9] := RETAINTEST_AUTO_STRUCTUREARRAYARRAY.ARRAYARRAY_INT[6][9];

    RETAINTEST_AUTO_STRUCTUREARRAYARRAY.ARRAYARRAY_LINT[0][0] := RETAINTEST_AUTO_STRUCTUREARRAYARRAY.ARRAYARRAY_LINT[0][0] + 1;
    RETAINTEST_AUTO_STRUCTUREARRAYARRAY.ARRAYARRAY_LINT[0][1] := RETAINTEST_AUTO_STRUCTUREARRAYARRAY.ARRAYARRAY_LINT[0][1] + 1;
    RETAINTEST_AUTO_STRUCTUREARRAYARRAY.ARRAYARRAY_LINT[0][2] := RETAINTEST_AUTO_STRUCTUREARRAYARRAY.ARRAYARRAY_LINT[0][2] + 1;
    RETAINTEST_AUTO_STRUCTUREARRAYARRAY.ARRAYARRAY_LINT[0][3] := RETAINTEST_AUTO_STRUCTUREARRAYARRAY.ARRAYARRAY_LINT[0][3] + 1;
    RETAINTEST_AUTO_STRUCTUREARRAYARRAY.ARRAYARRAY_LINT[0][4] := RETAINTEST_AUTO_STRUCTUREARRAYARRAY.ARRAYARRAY_LINT[0][4] + 1;
    RETAINTEST_AUTO_STRUCTUREARRAYARRAY.ARRAYARRAY_LINT[0][5] := RETAINTEST_AUTO_STRUCTUREARRAYARRAY.ARRAYARRAY_LINT[0][5] + 1;
    RETAINTEST_AUTO_STRUCTUREARRAYARRAY.ARRAYARRAY_LINT[0][6] := RETAINTEST_AUTO_STRUCTUREARRAYARRAY.ARRAYARRAY_LINT[0][6] + 1;
    RETAINTEST_AUTO_STRUCTUREARRAYARRAY.ARRAYARRAY_LINT[0][7] := RETAINTEST_AUTO_STRUCTUREARRAYARRAY.ARRAYARRAY_LINT[0][7] + 1;
    RETAINTEST_AUTO_STRUCTUREARRAYARRAY.ARRAYARRAY_LINT[0][8] := RETAINTEST_AUTO_STRUCTUREARRAYARRAY.ARRAYARRAY_LINT[0][6];
    RETAINTEST_AUTO_STRUCTUREARRAYARRAY.ARRAYARRAY_LINT[0][9] := RETAINTEST_AUTO_STRUCTUREARRAYARRAY.ARRAYARRAY_LINT[0][7];

    RETAINTEST_AUTO_STRUCTUREARRAYARRAY.ARRAYARRAY_LINT[1][0] := RETAINTEST_AUTO_STRUCTUREARRAYARRAY.ARRAYARRAY_LINT[1][0] + 1;
    RETAINTEST_AUTO_STRUCTUREARRAYARRAY.ARRAYARRAY_LINT[1][1] := RETAINTEST_AUTO_STRUCTUREARRAYARRAY.ARRAYARRAY_LINT[1][1] + 1;
    RETAINTEST_AUTO_STRUCTUREARRAYARRAY.ARRAYARRAY_LINT[1][2] := RETAINTEST_AUTO_STRUCTUREARRAYARRAY.ARRAYARRAY_LINT[1][2] + 1;
    RETAINTEST_AUTO_STRUCTUREARRAYARRAY.ARRAYARRAY_LINT[1][3] := RETAINTEST_AUTO_STRUCTUREARRAYARRAY.ARRAYARRAY_LINT[1][3] + 1;
    RETAINTEST_AUTO_STRUCTUREARRAYARRAY.ARRAYARRAY_LINT[1][4] := RETAINTEST_AUTO_STRUCTUREARRAYARRAY.ARRAYARRAY_LINT[1][4] + 1;
    RETAINTEST_AUTO_STRUCTUREARRAYARRAY.ARRAYARRAY_LINT[1][5] := RETAINTEST_AUTO_STRUCTUREARRAYARRAY.ARRAYARRAY_LINT[1][5] + 1;
    RETAINTEST_AUTO_STRUCTUREARRAYARRAY.ARRAYARRAY_LINT[1][6] := RETAINTEST_AUTO_STRUCTUREARRAYARRAY.ARRAYARRAY_LINT[1][6] + 1;
    RETAINTEST_AUTO_STRUCTUREARRAYARRAY.ARRAYARRAY_LINT[1][7] := RETAINTEST_AUTO_STRUCTUREARRAYARRAY.ARRAYARRAY_LINT[1][7] + 1;
    RETAINTEST_AUTO_STRUCTUREARRAYARRAY.ARRAYARRAY_LINT[1][8] := RETAINTEST_AUTO_STRUCTUREARRAYARRAY.ARRAYARRAY_LINT[1][6];
    RETAINTEST_AUTO_STRUCTUREARRAYARRAY.ARRAYARRAY_LINT[1][9] := RETAINTEST_AUTO_STRUCTUREARRAYARRAY.ARRAYARRAY_LINT[1][7];

    RETAINTEST_AUTO_STRUCTUREARRAYARRAY.ARRAYARRAY_LINT[2][0] := RETAINTEST_AUTO_STRUCTUREARRAYARRAY.ARRAYARRAY_LINT[2][0] + 1;
    RETAINTEST_AUTO_STRUCTUREARRAYARRAY.ARRAYARRAY_LINT[2][1] := RETAINTEST_AUTO_STRUCTUREARRAYARRAY.ARRAYARRAY_LINT[2][1] + 1;
    RETAINTEST_AUTO_STRUCTUREARRAYARRAY.ARRAYARRAY_LINT[2][2] := RETAINTEST_AUTO_STRUCTUREARRAYARRAY.ARRAYARRAY_LINT[2][2] + 1;
    RETAINTEST_AUTO_STRUCTUREARRAYARRAY.ARRAYARRAY_LINT[2][3] := RETAINTEST_AUTO_STRUCTUREARRAYARRAY.ARRAYARRAY_LINT[2][3] + 1;
    RETAINTEST_AUTO_STRUCTUREARRAYARRAY.ARRAYARRAY_LINT[2][4] := RETAINTEST_AUTO_STRUCTUREARRAYARRAY.ARRAYARRAY_LINT[2][4] + 1;
    RETAINTEST_AUTO_STRUCTUREARRAYARRAY.ARRAYARRAY_LINT[2][5] := RETAINTEST_AUTO_STRUCTUREARRAYARRAY.ARRAYARRAY_LINT[2][5] + 1;
    RETAINTEST_AUTO_STRUCTUREARRAYARRAY.ARRAYARRAY_LINT[2][6] := RETAINTEST_AUTO_STRUCTUREARRAYARRAY.ARRAYARRAY_LINT[2][6] + 1;
    RETAINTEST_AUTO_STRUCTUREARRAYARRAY.ARRAYARRAY_LINT[2][7] := RETAINTEST_AUTO_STRUCTUREARRAYARRAY.ARRAYARRAY_LINT[2][7] + 1;
    RETAINTEST_AUTO_STRUCTUREARRAYARRAY.ARRAYARRAY_LINT[2][8] := RETAINTEST_AUTO_STRUCTUREARRAYARRAY.ARRAYARRAY_LINT[2][8] + 1;
    RETAINTEST_AUTO_STRUCTUREARRAYARRAY.ARRAYARRAY_LINT[2][9] := RETAINTEST_AUTO_STRUCTUREARRAYARRAY.ARRAYARRAY_LINT[2][9] + 1;

    RETAINTEST_AUTO_STRUCTUREARRAYARRAY.ARRAYARRAY_LINT[3][0] := RETAINTEST_AUTO_STRUCTUREARRAYARRAY.ARRAYARRAY_LINT[3][0] + 1;
    RETAINTEST_AUTO_STRUCTUREARRAYARRAY.ARRAYARRAY_LINT[3][1] := RETAINTEST_AUTO_STRUCTUREARRAYARRAY.ARRAYARRAY_LINT[3][1] + 1;
    RETAINTEST_AUTO_STRUCTUREARRAYARRAY.ARRAYARRAY_LINT[3][2] := RETAINTEST_AUTO_STRUCTUREARRAYARRAY.ARRAYARRAY_LINT[3][2] + 1;
    RETAINTEST_AUTO_STRUCTUREARRAYARRAY.ARRAYARRAY_LINT[3][3] := RETAINTEST_AUTO_STRUCTUREARRAYARRAY.ARRAYARRAY_LINT[3][3] + 1;
    RETAINTEST_AUTO_STRUCTUREARRAYARRAY.ARRAYARRAY_LINT[3][4] := RETAINTEST_AUTO_STRUCTUREARRAYARRAY.ARRAYARRAY_LINT[3][4] + 1;
    RETAINTEST_AUTO_STRUCTUREARRAYARRAY.ARRAYARRAY_LINT[3][5] := RETAINTEST_AUTO_STRUCTUREARRAYARRAY.ARRAYARRAY_LINT[3][5] + 1;
    RETAINTEST_AUTO_STRUCTUREARRAYARRAY.ARRAYARRAY_LINT[3][6] := RETAINTEST_AUTO_STRUCTUREARRAYARRAY.ARRAYARRAY_LINT[3][6] + 1;
    RETAINTEST_AUTO_STRUCTUREARRAYARRAY.ARRAYARRAY_LINT[3][7] := RETAINTEST_AUTO_STRUCTUREARRAYARRAY.ARRAYARRAY_LINT[3][7] + 1;
    RETAINTEST_AUTO_STRUCTUREARRAYARRAY.ARRAYARRAY_LINT[3][8] := RETAINTEST_AUTO_STRUCTUREARRAYARRAY.ARRAYARRAY_LINT[3][8] + 1;
    RETAINTEST_AUTO_STRUCTUREARRAYARRAY.ARRAYARRAY_LINT[3][9] := RETAINTEST_AUTO_STRUCTUREARRAYARRAY.ARRAYARRAY_LINT[3][9] + 1;

    RETAINTEST_AUTO_STRUCTUREARRAYARRAY.ARRAYARRAY_LINT[4][0] := RETAINTEST_AUTO_STRUCTUREARRAYARRAY.ARRAYARRAY_LINT[4][0] + 1;
    RETAINTEST_AUTO_STRUCTUREARRAYARRAY.ARRAYARRAY_LINT[4][1] := RETAINTEST_AUTO_STRUCTUREARRAYARRAY.ARRAYARRAY_LINT[4][1] + 1;
    RETAINTEST_AUTO_STRUCTUREARRAYARRAY.ARRAYARRAY_LINT[4][2] := RETAINTEST_AUTO_STRUCTUREARRAYARRAY.ARRAYARRAY_LINT[4][2] + 1;
    RETAINTEST_AUTO_STRUCTUREARRAYARRAY.ARRAYARRAY_LINT[4][3] := RETAINTEST_AUTO_STRUCTUREARRAYARRAY.ARRAYARRAY_LINT[4][3] + 1;
    RETAINTEST_AUTO_STRUCTUREARRAYARRAY.ARRAYARRAY_LINT[4][4] := RETAINTEST_AUTO_STRUCTUREARRAYARRAY.ARRAYARRAY_LINT[4][4] + 1;
    RETAINTEST_AUTO_STRUCTUREARRAYARRAY.ARRAYARRAY_LINT[4][5] := RETAINTEST_AUTO_STRUCTUREARRAYARRAY.ARRAYARRAY_LINT[4][5] + 1;
    RETAINTEST_AUTO_STRUCTUREARRAYARRAY.ARRAYARRAY_LINT[4][6] := RETAINTEST_AUTO_STRUCTUREARRAYARRAY.ARRAYARRAY_LINT[4][6] + 1;
    RETAINTEST_AUTO_STRUCTUREARRAYARRAY.ARRAYARRAY_LINT[4][7] := RETAINTEST_AUTO_STRUCTUREARRAYARRAY.ARRAYARRAY_LINT[4][7] + 1;
    RETAINTEST_AUTO_STRUCTUREARRAYARRAY.ARRAYARRAY_LINT[4][8] := RETAINTEST_AUTO_STRUCTUREARRAYARRAY.ARRAYARRAY_LINT[4][8] + 1;
    RETAINTEST_AUTO_STRUCTUREARRAYARRAY.ARRAYARRAY_LINT[4][9] := RETAINTEST_AUTO_STRUCTUREARRAYARRAY.ARRAYARRAY_LINT[4][9] + 1;

    RETAINTEST_AUTO_STRUCTUREARRAYARRAY.ARRAYARRAY_LINT[5][0] := RETAINTEST_AUTO_STRUCTUREARRAYARRAY.ARRAYARRAY_LINT[5][0] + 1;
    RETAINTEST_AUTO_STRUCTUREARRAYARRAY.ARRAYARRAY_LINT[5][1] := RETAINTEST_AUTO_STRUCTUREARRAYARRAY.ARRAYARRAY_LINT[5][1] + 1;
    RETAINTEST_AUTO_STRUCTUREARRAYARRAY.ARRAYARRAY_LINT[5][2] := RETAINTEST_AUTO_STRUCTUREARRAYARRAY.ARRAYARRAY_LINT[5][2] + 1;
    RETAINTEST_AUTO_STRUCTUREARRAYARRAY.ARRAYARRAY_LINT[5][3] := RETAINTEST_AUTO_STRUCTUREARRAYARRAY.ARRAYARRAY_LINT[5][3] + 1;
    RETAINTEST_AUTO_STRUCTUREARRAYARRAY.ARRAYARRAY_LINT[5][4] := RETAINTEST_AUTO_STRUCTUREARRAYARRAY.ARRAYARRAY_LINT[5][4] + 1;
    RETAINTEST_AUTO_STRUCTUREARRAYARRAY.ARRAYARRAY_LINT[5][5] := RETAINTEST_AUTO_STRUCTUREARRAYARRAY.ARRAYARRAY_LINT[5][5] + 1;
    RETAINTEST_AUTO_STRUCTUREARRAYARRAY.ARRAYARRAY_LINT[5][6] := RETAINTEST_AUTO_STRUCTUREARRAYARRAY.ARRAYARRAY_LINT[5][6] + 1;
    RETAINTEST_AUTO_STRUCTUREARRAYARRAY.ARRAYARRAY_LINT[5][7] := RETAINTEST_AUTO_STRUCTUREARRAYARRAY.ARRAYARRAY_LINT[5][7] + 1;
    RETAINTEST_AUTO_STRUCTUREARRAYARRAY.ARRAYARRAY_LINT[5][8] := RETAINTEST_AUTO_STRUCTUREARRAYARRAY.ARRAYARRAY_LINT[5][8] + 1;
    RETAINTEST_AUTO_STRUCTUREARRAYARRAY.ARRAYARRAY_LINT[5][9] := RETAINTEST_AUTO_STRUCTUREARRAYARRAY.ARRAYARRAY_LINT[5][9] + 1;

    RETAINTEST_AUTO_STRUCTUREARRAYARRAY.ARRAYARRAY_LINT[6][0] := RETAINTEST_AUTO_STRUCTUREARRAYARRAY.ARRAYARRAY_LINT[6][0] + 1;
    RETAINTEST_AUTO_STRUCTUREARRAYARRAY.ARRAYARRAY_LINT[6][1] := RETAINTEST_AUTO_STRUCTUREARRAYARRAY.ARRAYARRAY_LINT[6][1] + 1;
    RETAINTEST_AUTO_STRUCTUREARRAYARRAY.ARRAYARRAY_LINT[6][2] := RETAINTEST_AUTO_STRUCTUREARRAYARRAY.ARRAYARRAY_LINT[6][2] + 1;
    RETAINTEST_AUTO_STRUCTUREARRAYARRAY.ARRAYARRAY_LINT[6][3] := RETAINTEST_AUTO_STRUCTUREARRAYARRAY.ARRAYARRAY_LINT[6][3] + 1;
    RETAINTEST_AUTO_STRUCTUREARRAYARRAY.ARRAYARRAY_LINT[6][4] := RETAINTEST_AUTO_STRUCTUREARRAYARRAY.ARRAYARRAY_LINT[6][4] + 1;
    RETAINTEST_AUTO_STRUCTUREARRAYARRAY.ARRAYARRAY_LINT[6][5] := RETAINTEST_AUTO_STRUCTUREARRAYARRAY.ARRAYARRAY_LINT[6][5] + 1;
    RETAINTEST_AUTO_STRUCTUREARRAYARRAY.ARRAYARRAY_LINT[6][6] := RETAINTEST_AUTO_STRUCTUREARRAYARRAY.ARRAYARRAY_LINT[6][6] + 1;
    RETAINTEST_AUTO_STRUCTUREARRAYARRAY.ARRAYARRAY_LINT[6][7] := RETAINTEST_AUTO_STRUCTUREARRAYARRAY.ARRAYARRAY_LINT[6][7] + 1;
    RETAINTEST_AUTO_STRUCTUREARRAYARRAY.ARRAYARRAY_LINT[6][8] := RETAINTEST_AUTO_STRUCTUREARRAYARRAY.ARRAYARRAY_LINT[6][8] + 1;
    RETAINTEST_AUTO_STRUCTUREARRAYARRAY.ARRAYARRAY_LINT[6][9] := RETAINTEST_AUTO_STRUCTUREARRAYARRAY.ARRAYARRAY_LINT[6][9] + 1;

    RETAINTEST_AUTO_STRUCTUREARRAYARRAY.ARRAYARRAY_LINT[7][0] := RETAINTEST_AUTO_STRUCTUREARRAYARRAY.ARRAYARRAY_LINT[6][0];
    RETAINTEST_AUTO_STRUCTUREARRAYARRAY.ARRAYARRAY_LINT[7][1] := RETAINTEST_AUTO_STRUCTUREARRAYARRAY.ARRAYARRAY_LINT[6][1];
    RETAINTEST_AUTO_STRUCTUREARRAYARRAY.ARRAYARRAY_LINT[7][2] := RETAINTEST_AUTO_STRUCTUREARRAYARRAY.ARRAYARRAY_LINT[6][2];
    RETAINTEST_AUTO_STRUCTUREARRAYARRAY.ARRAYARRAY_LINT[7][3] := RETAINTEST_AUTO_STRUCTUREARRAYARRAY.ARRAYARRAY_LINT[6][3];
    RETAINTEST_AUTO_STRUCTUREARRAYARRAY.ARRAYARRAY_LINT[7][4] := RETAINTEST_AUTO_STRUCTUREARRAYARRAY.ARRAYARRAY_LINT[6][4];
    RETAINTEST_AUTO_STRUCTUREARRAYARRAY.ARRAYARRAY_LINT[7][5] := RETAINTEST_AUTO_STRUCTUREARRAYARRAY.ARRAYARRAY_LINT[6][5];
    RETAINTEST_AUTO_STRUCTUREARRAYARRAY.ARRAYARRAY_LINT[7][6] := RETAINTEST_AUTO_STRUCTUREARRAYARRAY.ARRAYARRAY_LINT[6][6];
    RETAINTEST_AUTO_STRUCTUREARRAYARRAY.ARRAYARRAY_LINT[7][7] := RETAINTEST_AUTO_STRUCTUREARRAYARRAY.ARRAYARRAY_LINT[6][7];
    RETAINTEST_AUTO_STRUCTUREARRAYARRAY.ARRAYARRAY_LINT[7][8] := RETAINTEST_AUTO_STRUCTUREARRAYARRAY.ARRAYARRAY_LINT[6][8];
    RETAINTEST_AUTO_STRUCTUREARRAYARRAY.ARRAYARRAY_LINT[7][9] := RETAINTEST_AUTO_STRUCTUREARRAYARRAY.ARRAYARRAY_LINT[6][9];

    RETAINTEST_AUTO_STRUCTUREARRAYARRAY.ARRAYARRAY_LREAL[0][0] := RETAINTEST_AUTO_STRUCTUREARRAYARRAY.ARRAYARRAY_LREAL[0][0] + 1.1;
    RETAINTEST_AUTO_STRUCTUREARRAYARRAY.ARRAYARRAY_LREAL[0][1] := RETAINTEST_AUTO_STRUCTUREARRAYARRAY.ARRAYARRAY_LREAL[0][1] + 1.1;
    RETAINTEST_AUTO_STRUCTUREARRAYARRAY.ARRAYARRAY_LREAL[0][2] := RETAINTEST_AUTO_STRUCTUREARRAYARRAY.ARRAYARRAY_LREAL[0][2] + 1.1;
    RETAINTEST_AUTO_STRUCTUREARRAYARRAY.ARRAYARRAY_LREAL[0][3] := RETAINTEST_AUTO_STRUCTUREARRAYARRAY.ARRAYARRAY_LREAL[0][3] + 1.1;
    RETAINTEST_AUTO_STRUCTUREARRAYARRAY.ARRAYARRAY_LREAL[0][4] := RETAINTEST_AUTO_STRUCTUREARRAYARRAY.ARRAYARRAY_LREAL[0][4] + 1.1;
    RETAINTEST_AUTO_STRUCTUREARRAYARRAY.ARRAYARRAY_LREAL[0][5] := RETAINTEST_AUTO_STRUCTUREARRAYARRAY.ARRAYARRAY_LREAL[0][5] + 1.1;
    RETAINTEST_AUTO_STRUCTUREARRAYARRAY.ARRAYARRAY_LREAL[0][6] := RETAINTEST_AUTO_STRUCTUREARRAYARRAY.ARRAYARRAY_LREAL[0][6] + 1.1;
    RETAINTEST_AUTO_STRUCTUREARRAYARRAY.ARRAYARRAY_LREAL[0][7] := RETAINTEST_AUTO_STRUCTUREARRAYARRAY.ARRAYARRAY_LREAL[0][7] + 1.1;
    RETAINTEST_AUTO_STRUCTUREARRAYARRAY.ARRAYARRAY_LREAL[0][8] := RETAINTEST_AUTO_STRUCTUREARRAYARRAY.ARRAYARRAY_LREAL[0][6];
    RETAINTEST_AUTO_STRUCTUREARRAYARRAY.ARRAYARRAY_LREAL[0][9] := RETAINTEST_AUTO_STRUCTUREARRAYARRAY.ARRAYARRAY_LREAL[0][7];

    RETAINTEST_AUTO_STRUCTUREARRAYARRAY.ARRAYARRAY_LREAL[1][0] := RETAINTEST_AUTO_STRUCTUREARRAYARRAY.ARRAYARRAY_LREAL[1][0] + 1.1;
    RETAINTEST_AUTO_STRUCTUREARRAYARRAY.ARRAYARRAY_LREAL[1][1] := RETAINTEST_AUTO_STRUCTUREARRAYARRAY.ARRAYARRAY_LREAL[1][1] + 1.1;
    RETAINTEST_AUTO_STRUCTUREARRAYARRAY.ARRAYARRAY_LREAL[1][2] := RETAINTEST_AUTO_STRUCTUREARRAYARRAY.ARRAYARRAY_LREAL[1][2] + 1.1;
    RETAINTEST_AUTO_STRUCTUREARRAYARRAY.ARRAYARRAY_LREAL[1][3] := RETAINTEST_AUTO_STRUCTUREARRAYARRAY.ARRAYARRAY_LREAL[1][3] + 1.1;
    RETAINTEST_AUTO_STRUCTUREARRAYARRAY.ARRAYARRAY_LREAL[1][4] := RETAINTEST_AUTO_STRUCTUREARRAYARRAY.ARRAYARRAY_LREAL[1][4] + 1.1;
    RETAINTEST_AUTO_STRUCTUREARRAYARRAY.ARRAYARRAY_LREAL[1][5] := RETAINTEST_AUTO_STRUCTUREARRAYARRAY.ARRAYARRAY_LREAL[1][5] + 1.1;
    RETAINTEST_AUTO_STRUCTUREARRAYARRAY.ARRAYARRAY_LREAL[1][6] := RETAINTEST_AUTO_STRUCTUREARRAYARRAY.ARRAYARRAY_LREAL[1][6] + 1.1;
    RETAINTEST_AUTO_STRUCTUREARRAYARRAY.ARRAYARRAY_LREAL[1][7] := RETAINTEST_AUTO_STRUCTUREARRAYARRAY.ARRAYARRAY_LREAL[1][7] + 1.1;
    RETAINTEST_AUTO_STRUCTUREARRAYARRAY.ARRAYARRAY_LREAL[1][8] := RETAINTEST_AUTO_STRUCTUREARRAYARRAY.ARRAYARRAY_LREAL[1][6];
    RETAINTEST_AUTO_STRUCTUREARRAYARRAY.ARRAYARRAY_LREAL[1][9] := RETAINTEST_AUTO_STRUCTUREARRAYARRAY.ARRAYARRAY_LREAL[1][7];
